LIN {X 20.739,Y -41.059,Z -74.568,A -90.000,B 90.000,C 0.000} C_DIS
LIN {X 20.794,Y -41.067,Z -74.409,A -90.000,B 90.000,C 0.000} C_DIS
LIN {X 20.845,Y -41.076,Z -74.290,A -90.000,B 90.000,C 0.000} C_DIS
LIN {X 20.887,Y -41.080,Z -74.206,A -90.000,B 90.000,C 0.000} C_DIS
LIN {X 20.922,Y -41.083,Z -74.143,A -90.000,B 90.000,C 0.000} C_DIS
LIN {X 20.977,Y -41.084,Z -74.055,A -90.000,B 90.000,C 0.000} C_DIS
LIN {X 21.019,Y -41.085,Z -73.993,A -90.000,B 90.000,C 0.000} C_DIS
LIN {X 21.124,Y -41.081,Z -73.850,A -90.000,B 90.000,C 0.000} C_DIS
LIN {X 21.182,Y -41.076,Z -73.781,A -90.000,B 90.000,C 0.000} C_DIS
LIN {X 21.231,Y -41.072,Z -73.726,A -90.000,B 90.000,C 0.000} C_DIS
LIN {X 21.448,Y -41.048,Z -73.510,A -90.000,B 90.000,C 0.000} C_DIS
LIN {X 21.548,Y -41.035,Z -73.423,A -90.000,B 90.000,C 0.000} C_DIS
LIN {X 21.638,Y -41.027,Z -73.353,A -90.000,B 90.000,C 0.000} C_DIS
LIN {X 21.731,Y -41.021,Z -73.289,A -90.000,B 90.000,C 0.000} C_DIS
LIN {X 21.845,Y -41.016,Z -73.219,A -90.000,B 90.000,C 0.000} C_DIS
LIN {X 22.045,Y -41.002,Z -73.109,A -90.000,B 90.000,C 0.000} C_DIS
LIN {X 22.194,Y -40.983,Z -73.040,A -90.000,B 90.000,C 0.000} C_DIS
LIN {X 22.361,Y -40.964,Z -72.980,A -90.000,B 90.000,C 0.000} C_DIS
LIN {X 22.407,Y -40.959,Z -72.966,A -90.000,B 90.000,C 0.000} C_DIS
LIN {X 22.608,Y -40.941,Z -72.918,A -90.000,B 90.000,C 0.000} C_DIS
LIN {X 22.750,Y -40.923,Z -72.888,A -90.000,B 90.000,C 0.000} C_DIS
LIN {X 22.851,Y -40.911,Z -72.872,A -90.000,B 90.000,C 0.000} C_DIS
LIN {X 22.918,Y -40.901,Z -72.865,A -90.000,B 90.000,C 0.000} C_DIS
LIN {X 22.991,Y -40.890,Z -72.860,A -90.000,B 90.000,C 0.000} C_DIS
LIN {X 23.121,Y -40.871,Z -72.857,A -90.000,B 90.000,C 0.000} C_DIS
LIN {X 23.421,Y -40.816,Z -72.816,A -90.000,B 90.000,C 0.000} C_DIS
LIN {X 23.607,Y -40.785,Z -72.800,A -90.000,B 90.000,C 0.000} C_DIS
LIN {X 23.837,Y -40.743,Z -72.806,A -90.000,B 90.000,C 0.000} C_DIS
LIN {X 24.098,Y -40.703,Z -72.831,A -90.000,B 90.000,C 0.000} C_DIS
LIN {X 24.287,Y -40.682,Z -72.862,A -90.000,B 90.000,C 0.000} C_DIS
LIN {X 24.457,Y -40.670,Z -72.906,A -90.000,B 90.000,C 0.000} C_DIS
LIN {X 24.895,Y -40.649,Z -73.037,A -90.000,B 90.000,C 0.000} C_DIS
LIN {X 24.984,Y -40.642,Z -73.064,A -90.000,B 90.000,C 0.000} C_DIS
LIN {X 25.233,Y -40.629,Z -73.149,A -90.000,B 90.000,C 0.000} C_DIS
LIN {X 25.886,Y -40.603,Z -73.389,A -90.000,B 90.000,C 0.000} C_DIS
LIN {X 26.129,Y -40.642,Z -73.460,A -90.000,B 90.000,C 0.000} C_DIS
LIN {X 26.235,Y -40.654,Z -73.492,A -90.000,B 90.000,C 0.000} C_DIS
LIN {X 26.356,Y -40.664,Z -73.532,A -90.000,B 90.000,C 0.000} C_DIS
LIN {X 26.477,Y -40.671,Z -73.577,A -90.000,B 90.000,C 0.000} C_DIS
LIN {X 26.624,Y -40.675,Z -73.643,A -90.000,B 90.000,C 0.000} C_DIS
LIN {X 26.712,Y -40.674,Z -73.692,A -90.000,B 90.000,C 0.000} C_DIS
LIN {X 26.777,Y -40.673,Z -73.731,A -90.000,B 90.000,C 0.000} C_DIS
LIN {X 27.152,Y -40.658,Z -73.985,A -90.000,B 90.000,C 0.000} C_DIS
LIN {X 27.234,Y -40.655,Z -74.042,A -90.000,B 90.000,C 0.000} C_DIS
LIN {X 27.334,Y -40.665,Z -74.106,A -90.000,B 90.000,C 0.000} C_DIS
LIN {X 27.515,Y -40.693,Z -74.240,A -90.000,B 90.000,C 0.000} C_DIS
LIN {X 27.742,Y -40.737,Z -74.427,A -90.000,B 90.000,C 0.000} C_DIS
LIN {X 28.067,Y -40.769,Z -74.619,A -90.000,B 90.000,C 0.000} C_DIS
LIN {X 28.270,Y -40.787,Z -74.741,A -90.000,B 90.000,C 0.000} C_DIS
LIN {X 28.484,Y -40.804,Z -74.883,A -90.000,B 90.000,C 0.000} C_DIS
LIN {X 28.589,Y -40.816,Z -74.962,A -90.000,B 90.000,C 0.000} C_DIS
LIN {X 28.701,Y -40.830,Z -75.051,A -90.000,B 90.000,C 0.000} C_DIS
LIN {X 28.816,Y -40.850,Z -75.156,A -90.000,B 90.000,C 0.000} C_DIS
LIN {X 28.899,Y -40.868,Z -75.243,A -90.000,B 90.000,C 0.000} C_DIS
LIN {X 29.007,Y -40.894,Z -75.364,A -90.000,B 90.000,C 0.000} C_DIS
LIN {X 29.056,Y -40.902,Z -75.422,A -90.000,B 90.000,C 0.000} C_DIS
LIN {X 29.140,Y -40.918,Z -75.531,A -90.000,B 90.000,C 0.000} C_DIS
LIN {X 29.065,Y -40.889,Z -75.375,A -90.000,B 90.000,C 0.000} C_DIS
LIN {X 29.035,Y -40.867,Z -75.304,A -90.000,B 90.000,C 0.000} C_DIS
LIN {X 28.987,Y -40.823,Z -75.163,A -90.000,B 90.000,C 0.000} C_DIS
LIN {X 28.912,Y -40.733,Z -74.888,A -90.000,B 90.000,C 0.000} C_DIS
LIN {X 28.896,Y -40.706,Z -74.820,A -90.000,B 90.000,C 0.000} C_DIS
LIN {X 28.875,Y -40.655,Z -74.711,A -90.000,B 90.000,C 0.000} C_DIS
LIN {X 28.863,Y -40.607,Z -74.612,A -90.000,B 90.000,C 0.000} C_DIS
LIN {X 28.857,Y -40.573,Z -74.542,A -90.000,B 90.000,C 0.000} C_DIS
LIN {X 28.785,Y -40.606,Z -74.333,A -90.000,B 90.000,C 0.000} C_DIS
LIN {X 28.697,Y -40.642,Z -74.065,A -90.000,B 90.000,C 0.000} C_DIS
LIN {X 28.660,Y -40.658,Z -73.938,A -90.000,B 90.000,C 0.000} C_DIS
LIN {X 28.633,Y -40.670,Z -73.800,A -90.000,B 90.000,C 0.000} C_DIS
LIN {X 28.563,Y -40.700,Z -73.393,A -90.000,B 90.000,C 0.000} C_DIS
LIN {X 28.554,Y -40.704,Z -73.311,A -90.000,B 90.000,C 0.000} C_DIS
LIN {X 28.534,Y -40.707,Z -73.108,A -90.000,B 90.000,C 0.000} C_DIS
LIN {X 28.507,Y -40.700,Z -72.788,A -90.000,B 90.000,C 0.000} C_DIS
LIN {X 28.500,Y -40.696,Z -72.665,A -90.000,B 90.000,C 0.000} C_DIS
LIN {X 28.496,Y -40.692,Z -72.535,A -90.000,B 90.000,C 0.000} C_DIS
LIN {X 28.495,Y -40.688,Z -72.486,A -90.000,B 90.000,C 0.000} C_DIS
LIN {X 28.495,Y -40.679,Z -72.413,A -90.000,B 90.000,C 0.000} C_DIS
LIN {X 28.493,Y -40.678,Z -72.374,A -90.000,B 90.000,C 0.000} C_DIS
LIN {X 28.493,Y -40.673,Z -72.333,A -90.000,B 90.000,C 0.000} C_DIS
LIN {X 28.491,Y -40.602,Z -71.772,A -90.000,B 90.000,C 0.000} C_DIS
LIN {X 28.496,Y -40.578,Z -71.671,A -90.000,B 90.000,C 0.000} C_DIS
LIN {X 28.513,Y -40.524,Z -71.446,A -90.000,B 90.000,C 0.000} C_DIS
LIN {X 28.522,Y -40.503,Z -71.363,A -90.000,B 90.000,C 0.000} C_DIS
LIN {X 28.535,Y -40.479,Z -71.269,A -90.000,B 90.000,C 0.000} C_DIS
LIN {X 28.558,Y -40.435,Z -71.147,A -90.000,B 90.000,C 0.000} C_DIS
LIN {X 28.608,Y -40.348,Z -70.924,A -90.000,B 90.000,C 0.000} C_DIS
LIN {X 28.637,Y -40.307,Z -70.822,A -90.000,B 90.000,C 0.000} C_DIS
LIN {X 28.684,Y -40.248,Z -70.684,A -90.000,B 90.000,C 0.000} C_DIS
LIN {X 28.761,Y -40.153,Z -70.522,A -90.000,B 90.000,C 0.000} C_DIS
LIN {X 28.872,Y -40.031,Z -70.321,A -90.000,B 90.000,C 0.000} C_DIS
LIN {X 28.886,Y -40.016,Z -70.298,A -90.000,B 90.000,C 0.000} C_DIS
LIN {X 28.903,Y -39.999,Z -70.278,A -90.000,B 90.000,C 0.000} C_DIS
LIN {X 28.971,Y -39.931,Z -70.206,A -90.000,B 90.000,C 0.000} C_DIS
LIN {X 29.041,Y -39.869,Z -70.144,A -90.000,B 90.000,C 0.000} C_DIS
LIN {X 29.042,Y -39.892,Z -69.943,A -90.000,B 90.000,C 0.000} C_DIS
LIN {X 29.046,Y -39.912,Z -69.756,A -90.000,B 90.000,C 0.000} C_DIS
LIN {X 29.061,Y -39.961,Z -69.383,A -90.000,B 90.000,C 0.000} C_DIS
LIN {X 29.065,Y -39.977,Z -69.251,A -90.000,B 90.000,C 0.000} C_DIS
LIN {X 29.040,Y -39.961,Z -69.052,A -90.000,B 90.000,C 0.000} C_DIS
LIN {X 29.024,Y -39.953,Z -68.893,A -90.000,B 90.000,C 0.000} C_DIS
LIN {X 29.017,Y -39.952,Z -68.804,A -90.000,B 90.000,C 0.000} C_DIS
LIN {X 29.002,Y -39.952,Z -68.566,A -90.000,B 90.000,C 0.000} C_DIS
LIN {X 28.985,Y -39.943,Z -68.293,A -90.000,B 90.000,C 0.000} C_DIS
LIN {X 28.973,Y -39.937,Z -68.071,A -90.000,B 90.000,C 0.000} C_DIS
LIN {X 28.934,Y -39.926,Z -67.437,A -90.000,B 90.000,C 0.000} C_DIS
LIN {X 28.921,Y -39.924,Z -67.208,A -90.000,B 90.000,C 0.000} C_DIS
LIN {X 28.917,Y -39.922,Z -67.103,A -90.000,B 90.000,C 0.000} C_DIS
LIN {X 28.915,Y -39.923,Z -66.972,A -90.000,B 90.000,C 0.000} C_DIS
LIN {X 28.917,Y -39.946,Z -66.272,A -90.000,B 90.000,C 0.000} C_DIS
LIN {X 28.925,Y -39.969,Z -65.802,A -90.000,B 90.000,C 0.000} C_DIS
LIN {X 28.936,Y -39.980,Z -65.477,A -90.000,B 90.000,C 0.000} C_DIS
LIN {X 28.952,Y -39.998,Z -65.100,A -90.000,B 90.000,C 0.000} C_DIS
LIN {X 28.961,Y -40.008,Z -64.964,A -90.000,B 90.000,C 0.000} C_DIS
LIN {X 28.991,Y -40.040,Z -64.705,A -90.000,B 90.000,C 0.000} C_DIS
LIN {X 29.056,Y -40.094,Z -64.224,A -90.000,B 90.000,C 0.000} C_DIS
LIN {X 29.097,Y -40.123,Z -63.947,A -90.000,B 90.000,C 0.000} C_DIS
LIN {X 29.164,Y -40.154,Z -63.594,A -90.000,B 90.000,C 0.000} C_DIS
LIN {X 29.181,Y -40.164,Z -63.517,A -90.000,B 90.000,C 0.000} C_DIS
LIN {X 29.246,Y -40.202,Z -63.255,A -90.000,B 90.000,C 0.000} C_DIS
LIN {X 29.278,Y -40.220,Z -63.112,A -90.000,B 90.000,C 0.000} C_DIS
LIN {X 29.318,Y -40.233,Z -62.982,A -90.000,B 90.000,C 0.000} C_DIS
LIN {X 29.371,Y -40.252,Z -62.818,A -90.000,B 90.000,C 0.000} C_DIS
LIN {X 29.470,Y -40.290,Z -62.526,A -90.000,B 90.000,C 0.000} C_DIS
LIN {X 29.513,Y -40.308,Z -62.410,A -90.000,B 90.000,C 0.000} C_DIS
LIN {X 29.558,Y -40.330,Z -62.304,A -90.000,B 90.000,C 0.000} C_DIS
LIN {X 29.722,Y -40.380,Z -61.991,A -90.000,B 90.000,C 0.000} C_DIS
LIN {X 29.790,Y -40.400,Z -61.875,A -90.000,B 90.000,C 0.000} C_DIS
LIN {X 29.906,Y -40.431,Z -61.702,A -90.000,B 90.000,C 0.000} C_DIS
LIN {X 30.022,Y -40.458,Z -61.534,A -90.000,B 90.000,C 0.000} C_DIS
LIN {X 30.098,Y -40.470,Z -61.437,A -90.000,B 90.000,C 0.000} C_DIS
LIN {X 30.199,Y -40.487,Z -61.317,A -90.000,B 90.000,C 0.000} C_DIS
LIN {X 30.265,Y -40.494,Z -61.242,A -90.000,B 90.000,C 0.000} C_DIS
LIN {X 30.445,Y -40.400,Z -60.703,A -90.000,B 90.000,C 0.000} C_DIS
LIN {X 30.536,Y -40.349,Z -60.445,A -90.000,B 90.000,C 0.000} C_DIS
LIN {X 30.632,Y -40.305,Z -60.205,A -90.000,B 90.000,C 0.000} C_DIS
LIN {X 30.748,Y -40.248,Z -59.942,A -90.000,B 90.000,C 0.000} C_DIS
LIN {X 30.826,Y -40.210,Z -59.773,A -90.000,B 90.000,C 0.000} C_DIS
LIN {X 30.903,Y -40.172,Z -59.615,A -90.000,B 90.000,C 0.000} C_DIS
LIN {X 30.938,Y -40.153,Z -59.545,A -90.000,B 90.000,C 0.000} C_DIS
LIN {X 31.044,Y -40.095,Z -59.356,A -90.000,B 90.000,C 0.000} C_DIS
LIN {X 31.169,Y -40.028,Z -59.149,A -90.000,B 90.000,C 0.000} C_DIS
LIN {X 31.259,Y -39.978,Z -59.017,A -90.000,B 90.000,C 0.000} C_DIS
LIN {X 31.430,Y -39.885,Z -58.777,A -90.000,B 90.000,C 0.000} C_DIS
LIN {X 31.622,Y -39.782,Z -58.547,A -90.000,B 90.000,C 0.000} C_DIS
LIN {X 31.743,Y -39.722,Z -58.414,A -90.000,B 90.000,C 0.000} C_DIS
LIN {X 31.849,Y -39.675,Z -58.309,A -90.000,B 90.000,C 0.000} C_DIS
LIN {X 31.940,Y -39.637,Z -58.230,A -90.000,B 90.000,C 0.000} C_DIS
LIN {X 32.000,Y -39.612,Z -58.182,A -90.000,B 90.000,C 0.000} C_DIS
LIN {X 32.051,Y -39.624,Z -57.993,A -90.000,B 90.000,C 0.000} C_DIS
LIN {X 32.124,Y -39.645,Z -57.729,A -90.000,B 90.000,C 0.000} C_DIS
LIN {X 32.237,Y -39.661,Z -57.406,A -90.000,B 90.000,C 0.000} C_DIS
LIN {X 32.279,Y -39.668,Z -57.289,A -90.000,B 90.000,C 0.000} C_DIS
LIN {X 32.419,Y -39.706,Z -56.914,A -90.000,B 90.000,C 0.000} C_DIS
LIN {X 32.507,Y -39.732,Z -56.679,A -90.000,B 90.000,C 0.000} C_DIS
LIN {X 32.616,Y -39.765,Z -56.387,A -90.000,B 90.000,C 0.000} C_DIS
LIN {X 32.780,Y -39.791,Z -56.009,A -90.000,B 90.000,C 0.000} C_DIS
LIN {X 32.795,Y -39.792,Z -55.977,A -90.000,B 90.000,C 0.000} C_DIS
LIN {X 32.962,Y -39.810,Z -55.645,A -90.000,B 90.000,C 0.000} C_DIS
LIN {X 33.054,Y -39.815,Z -55.481,A -90.000,B 90.000,C 0.000} C_DIS
LIN {X 33.192,Y -39.830,Z -55.249,A -90.000,B 90.000,C 0.000} C_DIS
LIN {X 33.254,Y -39.840,Z -55.140,A -90.000,B 90.000,C 0.000} C_DIS
LIN {X 33.328,Y -39.853,Z -55.016,A -90.000,B 90.000,C 0.000} C_DIS
LIN {X 33.395,Y -39.866,Z -54.907,A -90.000,B 90.000,C 0.000} C_DIS
LIN {X 33.569,Y -39.902,Z -54.644,A -90.000,B 90.000,C 0.000} C_DIS
LIN {X 33.738,Y -39.918,Z -54.422,A -90.000,B 90.000,C 0.000} C_DIS
LIN {X 33.790,Y -39.921,Z -54.349,A -90.000,B 90.000,C 0.000} C_DIS
LIN {X 33.978,Y -39.939,Z -54.105,A -90.000,B 90.000,C 0.000} C_DIS
LIN {X 34.106,Y -39.942,Z -53.956,A -90.000,B 90.000,C 0.000} C_DIS
LIN {X 34.227,Y -39.950,Z -53.825,A -90.000,B 90.000,C 0.000} C_DIS
LIN {X 34.393,Y -39.967,Z -53.656,A -90.000,B 90.000,C 0.000} C_DIS
LIN {X 34.458,Y -39.977,Z -53.586,A -90.000,B 90.000,C 0.000} C_DIS
LIN {X 34.610,Y -39.992,Z -53.434,A -90.000,B 90.000,C 0.000} C_DIS
LIN {X 34.752,Y -40.008,Z -53.298,A -90.000,B 90.000,C 0.000} C_DIS
LIN {X 34.881,Y -40.012,Z -53.188,A -90.000,B 90.000,C 0.000} C_DIS
LIN {X 35.056,Y -40.015,Z -53.038,A -90.000,B 90.000,C 0.000} C_DIS
LIN {X 35.286,Y -40.009,Z -52.849,A -90.000,B 90.000,C 0.000} C_DIS
LIN {X 35.372,Y -40.009,Z -52.781,A -90.000,B 90.000,C 0.000} C_DIS
LIN {X 35.531,Y -40.015,Z -52.664,A -90.000,B 90.000,C 0.000} C_DIS
LIN {X 35.642,Y -40.023,Z -52.579,A -90.000,B 90.000,C 0.000} C_DIS
LIN {X 35.671,Y -40.025,Z -52.557,A -90.000,B 90.000,C 0.000} C_DIS
LIN {X 35.763,Y -40.025,Z -52.495,A -90.000,B 90.000,C 0.000} C_DIS
LIN {X 35.882,Y -40.031,Z -52.421,A -90.000,B 90.000,C 0.000} C_DIS
LIN {X 36.011,Y -40.041,Z -52.346,A -90.000,B 90.000,C 0.000} C_DIS
LIN {X 36.370,Y -40.043,Z -52.163,A -90.000,B 90.000,C 0.000} C_DIS
LIN {X 36.876,Y -40.035,Z -51.920,A -90.000,B 90.000,C 0.000} C_DIS
LIN {X 37.014,Y -40.034,Z -51.853,A -90.000,B 90.000,C 0.000} C_DIS
LIN {X 37.118,Y -40.036,Z -51.804,A -90.000,B 90.000,C 0.000} C_DIS
LIN {X 37.496,Y -40.037,Z -51.667,A -90.000,B 90.000,C 0.000} C_DIS
LIN {X 37.531,Y -40.035,Z -51.656,A -90.000,B 90.000,C 0.000} C_DIS
LIN {X 37.760,Y -40.029,Z -51.596,A -90.000,B 90.000,C 0.000} C_DIS
LIN {X 37.885,Y -40.030,Z -51.568,A -90.000,B 90.000,C 0.000} C_DIS
LIN {X 38.118,Y -40.025,Z -51.523,A -90.000,B 90.000,C 0.000} C_DIS
LIN {X 38.467,Y -40.023,Z -51.460,A -90.000,B 90.000,C 0.000} C_DIS
LIN {X 38.781,Y -40.023,Z -51.405,A -90.000,B 90.000,C 0.000} C_DIS
LIN {X 38.981,Y -40.016,Z -51.377,A -90.000,B 90.000,C 0.000} C_DIS
LIN {X 39.176,Y -40.011,Z -51.350,A -90.000,B 90.000,C 0.000} C_DIS
LIN {X 39.568,Y -39.990,Z -51.337,A -90.000,B 90.000,C 0.000} C_DIS
LIN {X 39.615,Y -39.985,Z -51.337,A -90.000,B 90.000,C 0.000} C_DIS
LIN {X 39.826,Y -39.975,Z -51.345,A -90.000,B 90.000,C 0.000} C_DIS
LIN {X 40.191,Y -39.968,Z -51.370,A -90.000,B 90.000,C 0.000} C_DIS
LIN {X 40.277,Y -39.968,Z -51.378,A -90.000,B 90.000,C 0.000} C_DIS
LIN {X 40.534,Y -39.973,Z -51.405,A -90.000,B 90.000,C 0.000} C_DIS
LIN {X 41.084,Y -39.977,Z -51.468,A -90.000,B 90.000,C 0.000} C_DIS
LIN {X 41.333,Y -39.964,Z -51.510,A -90.000,B 90.000,C 0.000} C_DIS
LIN {X 41.488,Y -39.958,Z -51.538,A -90.000,B 90.000,C 0.000} C_DIS
LIN {X 41.818,Y -39.925,Z -51.619,A -90.000,B 90.000,C 0.000} C_DIS
LIN {X 41.982,Y -39.914,Z -51.665,A -90.000,B 90.000,C 0.000} C_DIS
LIN {X 42.309,Y -39.902,Z -51.767,A -90.000,B 90.000,C 0.000} C_DIS
LIN {X 42.366,Y -39.899,Z -51.786,A -90.000,B 90.000,C 0.000} C_DIS
LIN {X 42.524,Y -39.895,Z -51.844,A -90.000,B 90.000,C 0.000} C_DIS
LIN {X 42.767,Y -39.896,Z -51.941,A -90.000,B 90.000,C 0.000} C_DIS
LIN {X 42.994,Y -39.896,Z -52.034,A -90.000,B 90.000,C 0.000} C_DIS
LIN {X 43.316,Y -39.884,Z -52.180,A -90.000,B 90.000,C 0.000} C_DIS
LIN {X 44.072,Y -39.861,Z -52.532,A -90.000,B 90.000,C 0.000} C_DIS
LIN {X 44.285,Y -39.859,Z -52.637,A -90.000,B 90.000,C 0.000} C_DIS
LIN {X 44.360,Y -39.858,Z -52.676,A -90.000,B 90.000,C 0.000} C_DIS
LIN {X 44.589,Y -39.862,Z -52.784,A -90.000,B 90.000,C 0.000} C_DIS
LIN {X 44.667,Y -39.865,Z -52.822,A -90.000,B 90.000,C 0.000} C_DIS
LIN {X 45.073,Y -39.887,Z -53.030,A -90.000,B 90.000,C 0.000} C_DIS
LIN {X 45.289,Y -39.893,Z -53.147,A -90.000,B 90.000,C 0.000} C_DIS
LIN {X 45.630,Y -39.938,Z -53.295,A -90.000,B 90.000,C 0.000} C_DIS
LIN {X 45.753,Y -39.958,Z -53.355,A -90.000,B 90.000,C 0.000} C_DIS
LIN {X 45.891,Y -40.000,Z -53.405,A -90.000,B 90.000,C 0.000} C_DIS
LIN {X 46.070,Y -40.052,Z -53.469,A -90.000,B 90.000,C 0.000} C_DIS
LIN {X 46.416,Y -40.159,Z -53.596,A -90.000,B 90.000,C 0.000} C_DIS
LIN {X 46.521,Y -40.196,Z -53.634,A -90.000,B 90.000,C 0.000} C_DIS
LIN {X 46.624,Y -40.202,Z -53.629,A -90.000,B 90.000,C 0.000} C_DIS
LIN {X 47.199,Y -40.201,Z -53.555,A -90.000,B 90.000,C 0.000} C_DIS
LIN {X 47.743,Y -40.204,Z -53.481,A -90.000,B 90.000,C 0.000} C_DIS
LIN {X 47.853,Y -40.203,Z -53.471,A -90.000,B 90.000,C 0.000} C_DIS
LIN {X 48.141,Y -40.205,Z -53.451,A -90.000,B 90.000,C 0.000} C_DIS
LIN {X 48.262,Y -40.202,Z -53.446,A -90.000,B 90.000,C 0.000} C_DIS
LIN {X 49.295,Y -40.205,Z -53.453,A -90.000,B 90.000,C 0.000} C_DIS
LIN {X 49.748,Y -40.210,Z -53.452,A -90.000,B 90.000,C 0.000} C_DIS
LIN {X 49.874,Y -40.208,Z -53.455,A -90.000,B 90.000,C 0.000} C_DIS
LIN {X 49.991,Y -40.207,Z -53.460,A -90.000,B 90.000,C 0.000} C_DIS
LIN {X 50.126,Y -40.208,Z -53.470,A -90.000,B 90.000,C 0.000} C_DIS
LIN {X 50.402,Y -40.194,Z -53.502,A -90.000,B 90.000,C 0.000} C_DIS
LIN {X 50.496,Y -40.192,Z -53.517,A -90.000,B 90.000,C 0.000} C_DIS
LIN {X 50.915,Y -40.174,Z -53.621,A -90.000,B 90.000,C 0.000} C_DIS
LIN {X 51.112,Y -40.173,Z -53.679,A -90.000,B 90.000,C 0.000} C_DIS
LIN {X 51.548,Y -40.185,Z -53.827,A -90.000,B 90.000,C 0.000} C_DIS
LIN {X 51.911,Y -40.190,Z -53.945,A -90.000,B 90.000,C 0.000} C_DIS
LIN {X 52.247,Y -40.200,Z -54.051,A -90.000,B 90.000,C 0.000} C_DIS
LIN {X 52.651,Y -40.202,Z -54.184,A -90.000,B 90.000,C 0.000} C_DIS
LIN {X 52.804,Y -40.191,Z -54.243,A -90.000,B 90.000,C 0.000} C_DIS
LIN {X 52.991,Y -40.182,Z -54.320,A -90.000,B 90.000,C 0.000} C_DIS
LIN {X 53.182,Y -40.162,Z -54.407,A -90.000,B 90.000,C 0.000} C_DIS
LIN {X 53.255,Y -40.156,Z -54.442,A -90.000,B 90.000,C 0.000} C_DIS
LIN {X 53.347,Y -40.152,Z -54.489,A -90.000,B 90.000,C 0.000} C_DIS
LIN {X 53.681,Y -40.126,Z -54.694,A -90.000,B 90.000,C 0.000} C_DIS
LIN {X 53.815,Y -40.120,Z -54.783,A -90.000,B 90.000,C 0.000} C_DIS
LIN {X 54.184,Y -40.113,Z -55.043,A -90.000,B 90.000,C 0.000} C_DIS
LIN {X 54.325,Y -40.115,Z -55.151,A -90.000,B 90.000,C 0.000} C_DIS
LIN {X 55.267,Y -40.165,Z -55.920,A -90.000,B 90.000,C 0.000} C_DIS
LIN {X 55.556,Y -40.166,Z -56.169,A -90.000,B 90.000,C 0.000} C_DIS
LIN {X 55.654,Y -40.159,Z -56.260,A -90.000,B 90.000,C 0.000} C_DIS
LIN {X 56.087,Y -40.112,Z -56.658,A -90.000,B 90.000,C 0.000} C_DIS
LIN {X 56.396,Y -40.082,Z -56.955,A -90.000,B 90.000,C 0.000} C_DIS
LIN {X 56.497,Y -40.075,Z -57.058,A -90.000,B 90.000,C 0.000} C_DIS
LIN {X 56.789,Y -40.071,Z -57.390,A -90.000,B 90.000,C 0.000} C_DIS
LIN {X 57.498,Y -40.083,Z -58.244,A -90.000,B 90.000,C 0.000} C_DIS
LIN {X 57.586,Y -40.088,Z -58.356,A -90.000,B 90.000,C 0.000} C_DIS
LIN {X 57.748,Y -40.101,Z -58.574,A -90.000,B 90.000,C 0.000} C_DIS
LIN {X 58.128,Y -40.098,Z -59.131,A -90.000,B 90.000,C 0.000} C_DIS
LIN {X 58.196,Y -40.099,Z -59.233,A -90.000,B 90.000,C 0.000} C_DIS
LIN {X 58.620,Y -40.116,Z -59.903,A -90.000,B 90.000,C 0.000} C_DIS
LIN {X 58.662,Y -40.119,Z -59.972,A -90.000,B 90.000,C 0.000} C_DIS
LIN {X 58.840,Y -40.136,Z -60.275,A -90.000,B 90.000,C 0.000} C_DIS
LIN {X 58.923,Y -40.146,Z -60.421,A -90.000,B 90.000,C 0.000} C_DIS
LIN {X 59.311,Y -40.200,Z -61.118,A -90.000,B 90.000,C 0.000} C_DIS
LIN {X 59.694,Y -40.209,Z -61.875,A -90.000,B 90.000,C 0.000} C_DIS
LIN {X 60.121,Y -40.201,Z -62.753,A -90.000,B 90.000,C 0.000} C_DIS
LIN {X 60.188,Y -40.203,Z -62.905,A -90.000,B 90.000,C 0.000} C_DIS
LIN {X 60.318,Y -40.217,Z -63.231,A -90.000,B 90.000,C 0.000} C_DIS
LIN {X 60.363,Y -40.224,Z -63.352,A -90.000,B 90.000,C 0.000} C_DIS
LIN {X 60.483,Y -40.252,Z -63.707,A -90.000,B 90.000,C 0.000} C_DIS
LIN {X 60.795,Y -40.313,Z -64.586,A -90.000,B 90.000,C 0.000} C_DIS
LIN {X 60.899,Y -40.321,Z -64.906,A -90.000,B 90.000,C 0.000} C_DIS
LIN {X 60.945,Y -40.321,Z -65.054,A -90.000,B 90.000,C 0.000} C_DIS
LIN {X 60.977,Y -40.318,Z -65.143,A -90.000,B 90.000,C 0.000} C_DIS
LIN {X 61.064,Y -40.318,Z -65.373,A -90.000,B 90.000,C 0.000} C_DIS
LIN {X 61.169,Y -40.325,Z -65.652,A -90.000,B 90.000,C 0.000} C_DIS
LIN {X 61.296,Y -40.341,Z -66.024,A -90.000,B 90.000,C 0.000} C_DIS
LIN {X 61.364,Y -40.358,Z -66.262,A -90.000,B 90.000,C 0.000} C_DIS
LIN {X 61.404,Y -40.375,Z -66.389,A -90.000,B 90.000,C 0.000} C_DIS
LIN {X 61.437,Y -40.392,Z -66.506,A -90.000,B 90.000,C 0.000} C_DIS
LIN {X 61.453,Y -40.404,Z -66.578,A -90.000,B 90.000,C 0.000} C_DIS
LIN {X 61.531,Y -40.476,Z -66.992,A -90.000,B 90.000,C 0.000} C_DIS
LIN {X 61.586,Y -40.495,Z -67.165,A -90.000,B 90.000,C 0.000} C_DIS
LIN {X 61.667,Y -40.510,Z -67.445,A -90.000,B 90.000,C 0.000} C_DIS
LIN {X 61.699,Y -40.513,Z -67.560,A -90.000,B 90.000,C 0.000} C_DIS
LIN {X 61.837,Y -40.496,Z -67.876,A -90.000,B 90.000,C 0.000} C_DIS
LIN {X 61.967,Y -40.504,Z -68.147,A -90.000,B 90.000,C 0.000} C_DIS
LIN {X 62.039,Y -40.513,Z -68.314,A -90.000,B 90.000,C 0.000} C_DIS
LIN {X 62.081,Y -40.524,Z -68.434,A -90.000,B 90.000,C 0.000} C_DIS
LIN {X 62.184,Y -40.557,Z -68.767,A -90.000,B 90.000,C 0.000} C_DIS
LIN {X 62.212,Y -40.570,Z -68.877,A -90.000,B 90.000,C 0.000} C_DIS
LIN {X 62.235,Y -40.594,Z -68.976,A -90.000,B 90.000,C 0.000} C_DIS
LIN {X 62.254,Y -40.619,Z -69.076,A -90.000,B 90.000,C 0.000} C_DIS
LIN {X 62.309,Y -40.686,Z -69.445,A -90.000,B 90.000,C 0.000} C_DIS
LIN {X 62.414,Y -40.703,Z -69.674,A -90.000,B 90.000,C 0.000} C_DIS
LIN {X 62.507,Y -40.705,Z -69.884,A -90.000,B 90.000,C 0.000} C_DIS
LIN {X 62.546,Y -40.702,Z -69.941,A -90.000,B 90.000,C 0.000} C_DIS
LIN {X 62.691,Y -40.685,Z -70.152,A -90.000,B 90.000,C 0.000} C_DIS
LIN {X 62.756,Y -40.680,Z -70.263,A -90.000,B 90.000,C 0.000} C_DIS
LIN {X 62.845,Y -40.673,Z -70.420,A -90.000,B 90.000,C 0.000} C_DIS
LIN {X 62.863,Y -40.675,Z -70.449,A -90.000,B 90.000,C 0.000} C_DIS
LIN {X 62.930,Y -40.686,Z -70.567,A -90.000,B 90.000,C 0.000} C_DIS
LIN {X 63.000,Y -40.702,Z -70.713,A -90.000,B 90.000,C 0.000} C_DIS
LIN {X 63.052,Y -40.720,Z -70.847,A -90.000,B 90.000,C 0.000} C_DIS
LIN {X 63.132,Y -40.750,Z -71.061,A -90.000,B 90.000,C 0.000} C_DIS
LIN {X 63.168,Y -40.767,Z -71.171,A -90.000,B 90.000,C 0.000} C_DIS
LIN {X 63.239,Y -40.802,Z -71.412,A -90.000,B 90.000,C 0.000} C_DIS
LIN {X 63.274,Y -40.828,Z -71.524,A -90.000,B 90.000,C 0.000} C_DIS
LIN {X 63.301,Y -40.854,Z -71.628,A -90.000,B 90.000,C 0.000} C_DIS
LIN {X 63.311,Y -40.863,Z -71.679,A -90.000,B 90.000,C 0.000} C_DIS
LIN {X 63.341,Y -40.893,Z -71.848,A -90.000,B 90.000,C 0.000} C_DIS
LIN {X 63.368,Y -40.935,Z -72.081,A -90.000,B 90.000,C 0.000} C_DIS
LIN {X 63.452,Y -40.946,Z -72.217,A -90.000,B 90.000,C 0.000} C_DIS
LIN {X 63.786,Y -40.929,Z -72.492,A -90.000,B 90.000,C 0.000} C_DIS
LIN {X 64.167,Y -40.899,Z -72.809,A -90.000,B 90.000,C 0.000} C_DIS
LIN {X 64.307,Y -40.889,Z -72.928,A -90.000,B 90.000,C 0.000} C_DIS
LIN {X 64.496,Y -40.878,Z -73.127,A -90.000,B 90.000,C 0.000} C_DIS
LIN {X 64.618,Y -40.888,Z -73.269,A -90.000,B 90.000,C 0.000} C_DIS
LIN {X 64.696,Y -40.895,Z -73.366,A -90.000,B 90.000,C 0.000} C_DIS
LIN {X 64.807,Y -40.900,Z -73.511,A -90.000,B 90.000,C 0.000} C_DIS
LIN {X 65.561,Y -40.793,Z -73.791,A -90.000,B 90.000,C 0.000} C_DIS
LIN {X 65.942,Y -40.738,Z -73.935,A -90.000,B 90.000,C 0.000} C_DIS
LIN {X 65.969,Y -40.737,Z -73.944,A -90.000,B 90.000,C 0.000} C_DIS
LIN {X 66.194,Y -40.728,Z -74.039,A -90.000,B 90.000,C 0.000} C_DIS
LIN {X 66.937,Y -40.714,Z -74.403,A -90.000,B 90.000,C 0.000} C_DIS
LIN {X 67.134,Y -40.704,Z -74.502,A -90.000,B 90.000,C 0.000} C_DIS
LIN {X 67.285,Y -40.696,Z -74.582,A -90.000,B 90.000,C 0.000} C_DIS
LIN {X 67.764,Y -40.679,Z -74.857,A -90.000,B 90.000,C 0.000} C_DIS
LIN {X 67.835,Y -40.677,Z -74.900,A -90.000,B 90.000,C 0.000} C_DIS
LIN {X 67.911,Y -40.676,Z -74.949,A -90.000,B 90.000,C 0.000} C_DIS
LIN {X 68.130,Y -40.678,Z -75.105,A -90.000,B 90.000,C 0.000} C_DIS
LIN {X 68.280,Y -40.682,Z -75.223,A -90.000,B 90.000,C 0.000} C_DIS
LIN {X 68.897,Y -40.724,Z -75.781,A -90.000,B 90.000,C 0.000} C_DIS
LIN {X 68.986,Y -40.724,Z -75.865,A -90.000,B 90.000,C 0.000} C_DIS
LIN {X 69.052,Y -40.732,Z -75.923,A -90.000,B 90.000,C 0.000} C_DIS
LIN {X 69.096,Y -40.730,Z -75.934,A -90.000,B 90.000,C 0.000} C_DIS
LIN {X 69.258,Y -40.709,Z -75.977,A -90.000,B 90.000,C 0.000} C_DIS
LIN {X 69.442,Y -40.681,Z -76.029,A -90.000,B 90.000,C 0.000} C_DIS
LIN {X 69.627,Y -40.654,Z -76.089,A -90.000,B 90.000,C 0.000} C_DIS
LIN {X 69.701,Y -40.643,Z -76.119,A -90.000,B 90.000,C 0.000} C_DIS
LIN {X 69.834,Y -40.625,Z -76.182,A -90.000,B 90.000,C 0.000} C_DIS
LIN {X 69.997,Y -40.597,Z -76.263,A -90.000,B 90.000,C 0.000} C_DIS
LIN {X 70.217,Y -40.565,Z -76.390,A -90.000,B 90.000,C 0.000} C_DIS
LIN {X 70.321,Y -40.555,Z -76.462,A -90.000,B 90.000,C 0.000} C_DIS
LIN {X 70.536,Y -40.535,Z -76.620,A -90.000,B 90.000,C 0.000} C_DIS
LIN {X 71.022,Y -40.539,Z -76.953,A -90.000,B 90.000,C 0.000} C_DIS
LIN {X 71.271,Y -40.552,Z -77.152,A -90.000,B 90.000,C 0.000} C_DIS
LIN {X 71.391,Y -40.557,Z -77.267,A -90.000,B 90.000,C 0.000} C_DIS
LIN {X 71.481,Y -40.563,Z -77.351,A -90.000,B 90.000,C 0.000} C_DIS
LIN {X 71.724,Y -40.572,Z -77.586,A -90.000,B 90.000,C 0.000} C_DIS
LIN {X 71.749,Y -40.569,Z -77.602,A -90.000,B 90.000,C 0.000} C_DIS
LIN {X 71.941,Y -40.541,Z -77.728,A -90.000,B 90.000,C 0.000} C_DIS
LIN {X 72.222,Y -40.507,Z -77.934,A -90.000,B 90.000,C 0.000} C_DIS
LIN {X 72.300,Y -40.499,Z -77.994,A -90.000,B 90.000,C 0.000} C_DIS
LIN {X 72.442,Y -40.488,Z -78.117,A -90.000,B 90.000,C 0.000} C_DIS
LIN {X 72.501,Y -40.478,Z -78.153,A -90.000,B 90.000,C 0.000} C_DIS
LIN {X 72.544,Y -40.475,Z -78.179,A -90.000,B 90.000,C 0.000} C_DIS
LIN {X 72.650,Y -40.470,Z -78.248,A -90.000,B 90.000,C 0.000} C_DIS
LIN {X 72.882,Y -40.463,Z -78.409,A -90.000,B 90.000,C 0.000} C_DIS
LIN {X 73.055,Y -40.464,Z -78.542,A -90.000,B 90.000,C 0.000} C_DIS
LIN {X 73.332,Y -40.466,Z -78.783,A -90.000,B 90.000,C 0.000} C_DIS
LIN {X 73.612,Y -40.461,Z -79.032,A -90.000,B 90.000,C 0.000} C_DIS
LIN {X 73.733,Y -40.458,Z -79.141,A -90.000,B 90.000,C 0.000} C_DIS
LIN {X 74.013,Y -40.437,Z -79.379,A -90.000,B 90.000,C 0.000} C_DIS
LIN {X 74.129,Y -40.431,Z -79.484,A -90.000,B 90.000,C 0.000} C_DIS
LIN {X 74.176,Y -40.433,Z -79.524,A -90.000,B 90.000,C 0.000} C_DIS
LIN {X 74.284,Y -40.429,Z -79.594,A -90.000,B 90.000,C 0.000} C_DIS
LIN {X 74.607,Y -40.420,Z -79.819,A -90.000,B 90.000,C 0.000} C_DIS
LIN {X 74.946,Y -40.411,Z -80.058,A -90.000,B 90.000,C 0.000} C_DIS
LIN {X 75.034,Y -40.411,Z -80.124,A -90.000,B 90.000,C 0.000} C_DIS
LIN {X 75.138,Y -40.410,Z -80.211,A -90.000,B 90.000,C 0.000} C_DIS
LIN {X 75.220,Y -40.404,Z -80.269,A -90.000,B 90.000,C 0.000} C_DIS
LIN {X 75.281,Y -40.402,Z -80.316,A -90.000,B 90.000,C 0.000} C_DIS
LIN {X 75.499,Y -40.423,Z -80.469,A -90.000,B 90.000,C 0.000} C_DIS
LIN {X 75.562,Y -40.423,Z -80.502,A -90.000,B 90.000,C 0.000} C_DIS
LIN {X 75.974,Y -40.440,Z -80.689,A -90.000,B 90.000,C 0.000} C_DIS
LIN {X 76.062,Y -40.438,Z -80.720,A -90.000,B 90.000,C 0.000} C_DIS
LIN {X 76.105,Y -40.434,Z -80.728,A -90.000,B 90.000,C 0.000} C_DIS
LIN {X 76.385,Y -40.404,Z -80.786,A -90.000,B 90.000,C 0.000} C_DIS
LIN {X 76.425,Y -40.395,Z -80.787,A -90.000,B 90.000,C 0.000} C_DIS
LIN {X 76.488,Y -40.387,Z -80.785,A -90.000,B 90.000,C 0.000} C_DIS
LIN {X 76.732,Y -40.368,Z -80.773,A -90.000,B 90.000,C 0.000} C_DIS
LIN {X 76.939,Y -40.369,Z -80.754,A -90.000,B 90.000,C 0.000} C_DIS
LIN {X 77.047,Y -40.363,Z -80.732,A -90.000,B 90.000,C 0.000} C_DIS
LIN {X 77.258,Y -40.347,Z -80.681,A -90.000,B 90.000,C 0.000} C_DIS
LIN {X 77.508,Y -40.321,Z -80.624,A -90.000,B 90.000,C 0.000} C_DIS
LIN {X 77.559,Y -40.319,Z -80.611,A -90.000,B 90.000,C 0.000} C_DIS
LIN {X 77.629,Y -40.318,Z -80.593,A -90.000,B 90.000,C 0.000} C_DIS
LIN {X 77.783,Y -40.310,Z -80.558,A -90.000,B 90.000,C 0.000} C_DIS
LIN {X 77.985,Y -40.303,Z -80.517,A -90.000,B 90.000,C 0.000} C_DIS
LIN {X 78.164,Y -40.298,Z -80.463,A -90.000,B 90.000,C 0.000} C_DIS
LIN {X 78.536,Y -40.279,Z -80.355,A -90.000,B 90.000,C 0.000} C_DIS
LIN {X 78.687,Y -40.277,Z -80.308,A -90.000,B 90.000,C 0.000} C_DIS
LIN {X 78.843,Y -40.269,Z -80.249,A -90.000,B 90.000,C 0.000} C_DIS
LIN {X 78.920,Y -40.263,Z -80.222,A -90.000,B 90.000,C 0.000} C_DIS
LIN {X 79.000,Y -40.175,Z -80.057,A -90.000,B 90.000,C 0.000} C_DIS
LIN {X 79.054,Y -40.118,Z -79.954,A -90.000,B 90.000,C 0.000} C_DIS
LIN {X 79.077,Y -40.084,Z -79.894,A -90.000,B 90.000,C 0.000} C_DIS
LIN {X 79.139,Y -39.998,Z -79.739,A -90.000,B 90.000,C 0.000} C_DIS
LIN {X 79.209,Y -39.913,Z -79.581,A -90.000,B 90.000,C 0.000} C_DIS
LIN {X 79.221,Y -39.897,Z -79.532,A -90.000,B 90.000,C 0.000} C_DIS
LIN {X 79.231,Y -39.884,Z -79.412,A -90.000,B 90.000,C 0.000} C_DIS
LIN {X 79.272,Y -39.838,Z -79.030,A -90.000,B 90.000,C 0.000} C_DIS
LIN {X 79.283,Y -39.829,Z -78.944,A -90.000,B 90.000,C 0.000} C_DIS
LIN {X 79.291,Y -39.827,Z -78.700,A -90.000,B 90.000,C 0.000} C_DIS
LIN {X 79.290,Y -39.812,Z -78.501,A -90.000,B 90.000,C 0.000} C_DIS
LIN {X 79.291,Y -39.785,Z -78.109,A -90.000,B 90.000,C 0.000} C_DIS
LIN {X 79.288,Y -39.781,Z -78.014,A -90.000,B 90.000,C 0.000} C_DIS
LIN {X 79.247,Y -39.732,Z -77.379,A -90.000,B 90.000,C 0.000} C_DIS
LIN {X 79.228,Y -39.723,Z -77.193,A -90.000,B 90.000,C 0.000} C_DIS
LIN {X 79.202,Y -39.708,Z -76.777,A -90.000,B 90.000,C 0.000} C_DIS
LIN {X 79.181,Y -39.695,Z -76.479,A -90.000,B 90.000,C 0.000} C_DIS
LIN {X 79.155,Y -39.667,Z -75.962,A -90.000,B 90.000,C 0.000} C_DIS
LIN {X 79.145,Y -39.663,Z -75.832,A -90.000,B 90.000,C 0.000} C_DIS
LIN {X 79.109,Y -39.641,Z -75.497,A -90.000,B 90.000,C 0.000} C_DIS
LIN {X 79.073,Y -39.620,Z -75.124,A -90.000,B 90.000,C 0.000} C_DIS
LIN {X 79.034,Y -39.607,Z -74.798,A -90.000,B 90.000,C 0.000} C_DIS
LIN {X 79.028,Y -39.603,Z -74.729,A -90.000,B 90.000,C 0.000} C_DIS
LIN {X 78.992,Y -39.585,Z -74.174,A -90.000,B 90.000,C 0.000} C_DIS
LIN {X 78.972,Y -39.561,Z -73.668,A -90.000,B 90.000,C 0.000} C_DIS
LIN {X 78.965,Y -39.553,Z -73.479,A -90.000,B 90.000,C 0.000} C_DIS
LIN {X 78.938,Y -39.518,Z -72.878,A -90.000,B 90.000,C 0.000} C_DIS
LIN {X 78.919,Y -39.494,Z -72.422,A -90.000,B 90.000,C 0.000} C_DIS
LIN {X 78.912,Y -39.485,Z -72.167,A -90.000,B 90.000,C 0.000} C_DIS
LIN {X 78.915,Y -39.468,Z -71.754,A -90.000,B 90.000,C 0.000} C_DIS
LIN {X 78.931,Y -39.453,Z -71.245,A -90.000,B 90.000,C 0.000} C_DIS
LIN {X 78.945,Y -39.446,Z -71.088,A -90.000,B 90.000,C 0.000} C_DIS
LIN {X 79.014,Y -39.419,Z -70.323,A -90.000,B 90.000,C 0.000} C_DIS
LIN {X 79.094,Y -39.395,Z -69.886,A -90.000,B 90.000,C 0.000} C_DIS
LIN {X 79.153,Y -39.380,Z -69.585,A -90.000,B 90.000,C 0.000} C_DIS
LIN {X 79.260,Y -39.360,Z -69.036,A -90.000,B 90.000,C 0.000} C_DIS
LIN {X 79.351,Y -39.348,Z -68.620,A -90.000,B 90.000,C 0.000} C_DIS
LIN {X 79.498,Y -39.334,Z -68.166,A -90.000,B 90.000,C 0.000} C_DIS
LIN {X 79.676,Y -39.324,Z -67.623,A -90.000,B 90.000,C 0.000} C_DIS
LIN {X 79.789,Y -39.318,Z -67.300,A -90.000,B 90.000,C 0.000} C_DIS
LIN {X 79.868,Y -39.316,Z -67.089,A -90.000,B 90.000,C 0.000} C_DIS
LIN {X 79.923,Y -39.315,Z -66.958,A -90.000,B 90.000,C 0.000} C_DIS
LIN {X 80.093,Y -39.311,Z -66.571,A -90.000,B 90.000,C 0.000} C_DIS
LIN {X 80.394,Y -39.309,Z -65.888,A -90.000,B 90.000,C 0.000} C_DIS
LIN {X 80.639,Y -39.309,Z -65.345,A -90.000,B 90.000,C 0.000} C_DIS
LIN {X 80.673,Y -39.309,Z -65.279,A -90.000,B 90.000,C 0.000} C_DIS
LIN {X 81.101,Y -39.317,Z -64.454,A -90.000,B 90.000,C 0.000} C_DIS
LIN {X 81.114,Y -39.320,Z -64.429,A -90.000,B 90.000,C 0.000} C_DIS
LIN {X 81.298,Y -39.318,Z -64.075,A -90.000,B 90.000,C 0.000} C_DIS
LIN {X 81.438,Y -39.308,Z -63.804,A -90.000,B 90.000,C 0.000} C_DIS
LIN {X 81.438,Y -60.000,Z -63.804,A -90.000,B 90.000,C 0.000} C_DIS
LIN {X 89.672,Y -60.000,Z -53.967,A -90.000,B 90.000,C 0.000} C_DIS
LIN {X 89.672,Y -39.308,Z -53.967,A -90.000,B 90.000,C 0.000} C_DIS
LIN {X 89.730,Y -39.308,Z -53.914,A -90.000,B 90.000,C 0.000} C_DIS
LIN {X 89.730,Y -60.000,Z -53.914,A -90.000,B 90.000,C 0.000} C_DIS
LIN {X 97.702,Y -60.000,Z -46.864,A -90.000,B 90.000,C 0.000} C_DIS
LIN {X 97.702,Y -39.308,Z -46.864,A -90.000,B 90.000,C 0.000} C_DIS
LIN {X 97.877,Y -39.308,Z -46.679,A -90.000,B 90.000,C 0.000} C_DIS
LIN {X 98.223,Y -44.514,Z -46.315,A -90.000,B 90.000,C 0.000} C_DIS
LIN {X 98.483,Y -44.409,Z -46.043,A -90.000,B 90.000,C 0.000} C_DIS
LIN {X 98.670,Y -44.352,Z -45.848,A -90.000,B 90.000,C 0.000} C_DIS
LIN {X 98.797,Y -44.328,Z -45.718,A -90.000,B 90.000,C 0.000} C_DIS
LIN {X 98.874,Y -44.327,Z -45.640,A -90.000,B 90.000,C 0.000} C_DIS
LIN {X 98.898,Y -44.332,Z -45.616,A -90.000,B 90.000,C 0.000} C_DIS
LIN {X 98.914,Y -44.339,Z -45.600,A -90.000,B 90.000,C 0.000} C_DIS
LIN {X 98.930,Y -44.355,Z -45.586,A -90.000,B 90.000,C 0.000} C_DIS
LIN {X 98.933,Y -44.368,Z -45.585,A -90.000,B 90.000,C 0.000} C_DIS
LIN {X 99.058,Y -44.166,Z -45.441,A -90.000,B 90.000,C 0.000} C_DIS
LIN {X 99.357,Y -43.911,Z -45.104,A -90.000,B 90.000,C 0.000} C_DIS
LIN {X 99.608,Y -43.722,Z -44.823,A -90.000,B 90.000,C 0.000} C_DIS
LIN {X 99.943,Y -39.308,Z -44.450,A -90.000,B 90.000,C 0.000} C_DIS
LIN {X 100.003,Y -39.310,Z -44.383,A -90.000,B 90.000,C 0.000} C_DIS
LIN {X 100.056,Y -39.308,Z -44.323,A -90.000,B 90.000,C 0.000} C_DIS
LIN {X 100.361,Y -43.219,Z -43.983,A -90.000,B 90.000,C 0.000} C_DIS
LIN {X 100.518,Y -43.132,Z -43.809,A -90.000,B 90.000,C 0.000} C_DIS
LIN {X 100.575,Y -43.094,Z -43.744,A -90.000,B 90.000,C 0.000} C_DIS
LIN {X 100.582,Y -43.085,Z -43.736,A -90.000,B 90.000,C 0.000} C_DIS
LIN {X 100.583,Y -43.066,Z -43.733,A -90.000,B 90.000,C 0.000} C_DIS
LIN {X 100.590,Y -43.049,Z -43.724,A -90.000,B 90.000,C 0.000} C_DIS
LIN {X 100.647,Y -42.983,Z -43.659,A -90.000,B 90.000,C 0.000} C_DIS
LIN {X 100.802,Y -42.848,Z -43.483,A -90.000,B 90.000,C 0.000} C_DIS
LIN {X 101.104,Y -39.308,Z -43.141,A -90.000,B 90.000,C 0.000} C_DIS
LIN {X 101.165,Y -39.308,Z -43.073,A -90.000,B 90.000,C 0.000} C_DIS
LIN {X 101.306,Y -42.474,Z -42.913,A -90.000,B 90.000,C 0.000} C_DIS
LIN {X 101.326,Y -42.463,Z -42.891,A -90.000,B 90.000,C 0.000} C_DIS
LIN {X 101.329,Y -42.473,Z -42.888,A -90.000,B 90.000,C 0.000} C_DIS
LIN {X 101.347,Y -42.474,Z -42.869,A -90.000,B 90.000,C 0.000} C_DIS
LIN {X 101.490,Y -39.308,Z -42.711,A -90.000,B 90.000,C 0.000} C_DIS
LIN {X 101.527,Y -39.308,Z -42.670,A -90.000,B 90.000,C 0.000} C_DIS
LIN {X 101.953,Y -41.785,Z -42.197,A -90.000,B 90.000,C 0.000} C_DIS
LIN {X 102.007,Y -41.721,Z -42.138,A -90.000,B 90.000,C 0.000} C_DIS
LIN {X 102.014,Y -41.732,Z -42.131,A -90.000,B 90.000,C 0.000} C_DIS
LIN {X 102.016,Y -41.778,Z -42.130,A -90.000,B 90.000,C 0.000} C_DIS
LIN {X 102.023,Y -41.796,Z -42.123,A -90.000,B 90.000,C 0.000} C_DIS
LIN {X 102.078,Y -41.787,Z -42.065,A -90.000,B 90.000,C 0.000} C_DIS
LIN {X 102.224,Y -41.679,Z -41.906,A -90.000,B 90.000,C 0.000} C_DIS
LIN {X 102.508,Y -39.308,Z -41.596,A -90.000,B 90.000,C 0.000} C_DIS
LIN {X 102.577,Y -39.308,Z -41.520,A -90.000,B 90.000,C 0.000} C_DIS
LIN {X 102.653,Y -41.243,Z -41.437,A -90.000,B 90.000,C 0.000} C_DIS
LIN {X 102.663,Y -41.229,Z -41.426,A -90.000,B 90.000,C 0.000} C_DIS
LIN {X 102.676,Y -41.250,Z -41.414,A -90.000,B 90.000,C 0.000} C_DIS
LIN {X 102.753,Y -39.308,Z -41.331,A -90.000,B 90.000,C 0.000} C_DIS
LIN {X 103.579,Y -39.309,Z -40.452,A -90.000,B 90.000,C 0.000} C_DIS
LIN {X 104.447,Y -39.313,Z -39.580,A -90.000,B 90.000,C 0.000} C_DIS
LIN {X 104.780,Y -39.317,Z -39.269,A -90.000,B 90.000,C 0.000} C_DIS
LIN {X 105.187,Y -39.325,Z -38.863,A -90.000,B 90.000,C 0.000} C_DIS
LIN {X 105.542,Y -39.332,Z -38.542,A -90.000,B 90.000,C 0.000} C_DIS
LIN {X 105.806,Y -39.339,Z -38.316,A -90.000,B 90.000,C 0.000} C_DIS
LIN {X 106.173,Y -39.352,Z -38.002,A -90.000,B 90.000,C 0.000} C_DIS
LIN {X 106.715,Y -39.370,Z -37.601,A -90.000,B 90.000,C 0.000} C_DIS
LIN {X 106.864,Y -39.375,Z -37.496,A -90.000,B 90.000,C 0.000} C_DIS
LIN {X 107.009,Y -39.378,Z -37.399,A -90.000,B 90.000,C 0.000} C_DIS
LIN {X 107.123,Y -39.382,Z -37.325,A -90.000,B 90.000,C 0.000} C_DIS
LIN {X 107.483,Y -39.396,Z -37.113,A -90.000,B 90.000,C 0.000} C_DIS
LIN {X 107.945,Y -39.407,Z -36.871,A -90.000,B 90.000,C 0.000} C_DIS
LIN {X 108.132,Y -39.412,Z -36.782,A -90.000,B 90.000,C 0.000} C_DIS
LIN {X 108.381,Y -39.423,Z -36.667,A -90.000,B 90.000,C 0.000} C_DIS
LIN {X 108.815,Y -39.427,Z -36.512,A -90.000,B 90.000,C 0.000} C_DIS
LIN {X 109.214,Y -39.441,Z -36.375,A -90.000,B 90.000,C 0.000} C_DIS
LIN {X 109.279,Y -39.441,Z -36.359,A -90.000,B 90.000,C 0.000} C_DIS
LIN {X 109.355,Y -39.442,Z -36.341,A -90.000,B 90.000,C 0.000} C_DIS
LIN {X 109.684,Y -39.454,Z -36.262,A -90.000,B 90.000,C 0.000} C_DIS
LIN {X 110.142,Y -39.456,Z -36.198,A -90.000,B 90.000,C 0.000} C_DIS
LIN {X 110.495,Y -39.466,Z -36.151,A -90.000,B 90.000,C 0.000} C_DIS
LIN {X 110.674,Y -39.468,Z -36.143,A -90.000,B 90.000,C 0.000} C_DIS
LIN {X 110.974,Y -39.476,Z -36.135,A -90.000,B 90.000,C 0.000} C_DIS
LIN {X 111.151,Y -39.476,Z -36.143,A -90.000,B 90.000,C 0.000} C_DIS
LIN {X 111.479,Y -39.477,Z -36.159,A -90.000,B 90.000,C 0.000} C_DIS
LIN {X 111.736,Y -39.485,Z -36.179,A -90.000,B 90.000,C 0.000} C_DIS
LIN {X 111.888,Y -39.486,Z -36.203,A -90.000,B 90.000,C 0.000} C_DIS
LIN {X 112.208,Y -39.492,Z -36.259,A -90.000,B 90.000,C 0.000} C_DIS
LIN {X 112.433,Y -39.494,Z -36.313,A -90.000,B 90.000,C 0.000} C_DIS
LIN {X 112.726,Y -39.495,Z -36.391,A -90.000,B 90.000,C 0.000} C_DIS
LIN {X 112.893,Y -39.501,Z -36.439,A -90.000,B 90.000,C 0.000} C_DIS
LIN {X 113.150,Y -39.504,Z -36.536,A -90.000,B 90.000,C 0.000} C_DIS
LIN {X 113.317,Y -39.507,Z -36.601,A -90.000,B 90.000,C 0.000} C_DIS
LIN {X 113.435,Y -39.514,Z -36.648,A -90.000,B 90.000,C 0.000} C_DIS
LIN {X 113.508,Y -39.516,Z -36.683,A -90.000,B 90.000,C 0.000} C_DIS
LIN {X 113.980,Y -39.524,Z -36.922,A -90.000,B 90.000,C 0.000} C_DIS
LIN {X 114.171,Y -39.534,Z -37.024,A -90.000,B 90.000,C 0.000} C_DIS
LIN {X 114.257,Y -39.537,Z -37.077,A -90.000,B 90.000,C 0.000} C_DIS
LIN {X 114.310,Y -39.540,Z -37.107,A -90.000,B 90.000,C 0.000} C_DIS
LIN {X 114.389,Y -39.542,Z -37.157,A -90.000,B 90.000,C 0.000} C_DIS
LIN {X 114.451,Y -39.545,Z -37.197,A -90.000,B 90.000,C 0.000} C_DIS
LIN {X 114.696,Y -39.565,Z -37.358,A -90.000,B 90.000,C 0.000} C_DIS
LIN {X 115.057,Y -39.580,Z -37.647,A -90.000,B 90.000,C 0.000} C_DIS
LIN {X 115.216,Y -39.583,Z -37.803,A -90.000,B 90.000,C 0.000} C_DIS
LIN {X 115.388,Y -39.590,Z -37.974,A -90.000,B 90.000,C 0.000} C_DIS
LIN {X 115.446,Y -39.589,Z -38.042,A -90.000,B 90.000,C 0.000} C_DIS
LIN {X 115.686,Y -39.599,Z -38.336,A -90.000,B 90.000,C 0.000} C_DIS
LIN {X 115.759,Y -39.599,Z -38.435,A -90.000,B 90.000,C 0.000} C_DIS
LIN {X 115.883,Y -39.605,Z -38.599,A -90.000,B 90.000,C 0.000} C_DIS
LIN {X 115.935,Y -39.605,Z -38.676,A -90.000,B 90.000,C 0.000} C_DIS
LIN {X 116.130,Y -39.614,Z -38.977,A -90.000,B 90.000,C 0.000} C_DIS
LIN {X 116.209,Y -39.613,Z -39.121,A -90.000,B 90.000,C 0.000} C_DIS
LIN {X 116.353,Y -39.617,Z -39.401,A -90.000,B 90.000,C 0.000} C_DIS
LIN {X 116.405,Y -39.615,Z -39.525,A -90.000,B 90.000,C 0.000} C_DIS
LIN {X 116.489,Y -39.617,Z -39.707,A -90.000,B 90.000,C 0.000} C_DIS
LIN {X 116.558,Y -39.615,Z -39.879,A -90.000,B 90.000,C 0.000} C_DIS
LIN {X 116.658,Y -39.621,Z -40.141,A -90.000,B 90.000,C 0.000} C_DIS
LIN {X 116.676,Y -39.619,Z -40.203,A -90.000,B 90.000,C 0.000} C_DIS
LIN {X 116.743,Y -39.618,Z -40.424,A -90.000,B 90.000,C 0.000} C_DIS
LIN {X 116.803,Y -39.615,Z -40.641,A -90.000,B 90.000,C 0.000} C_DIS
LIN {X 116.833,Y -39.616,Z -40.752,A -90.000,B 90.000,C 0.000} C_DIS
LIN {X 116.866,Y -39.622,Z -40.881,A -90.000,B 90.000,C 0.000} C_DIS
LIN {X 116.943,Y -39.617,Z -41.343,A -90.000,B 90.000,C 0.000} C_DIS
LIN {X 116.956,Y -39.615,Z -41.446,A -90.000,B 90.000,C 0.000} C_DIS
LIN {X 116.976,Y -39.618,Z -41.616,A -90.000,B 90.000,C 0.000} C_DIS
LIN {X 116.995,Y -39.617,Z -41.966,A -90.000,B 90.000,C 0.000} C_DIS
LIN {X 117.000,Y -39.619,Z -42.082,A -90.000,B 90.000,C 0.000} C_DIS
LIN {X 116.997,Y -39.616,Z -42.197,A -90.000,B 90.000,C 0.000} C_DIS
LIN {X 116.988,Y -39.613,Z -42.438,A -90.000,B 90.000,C 0.000} C_DIS
LIN {X 116.970,Y -39.614,Z -42.668,A -90.000,B 90.000,C 0.000} C_DIS
LIN {X 116.948,Y -39.611,Z -42.852,A -90.000,B 90.000,C 0.000} C_DIS
LIN {X 116.931,Y -39.611,Z -42.973,A -90.000,B 90.000,C 0.000} C_DIS
LIN {X 116.909,Y -39.617,Z -43.123,A -90.000,B 90.000,C 0.000} C_DIS
LIN {X 116.803,Y -39.612,Z -43.579,A -90.000,B 90.000,C 0.000} C_DIS
LIN {X 116.779,Y -39.610,Z -43.667,A -90.000,B 90.000,C 0.000} C_DIS
LIN {X 116.729,Y -39.614,Z -43.840,A -90.000,B 90.000,C 0.000} C_DIS
LIN {X 116.646,Y -39.613,Z -44.084,A -90.000,B 90.000,C 0.000} C_DIS
LIN {X 116.599,Y -39.616,Z -44.226,A -90.000,B 90.000,C 0.000} C_DIS
LIN {X 116.540,Y -39.625,Z -44.399,A -90.000,B 90.000,C 0.000} C_DIS
LIN {X 116.402,Y -39.658,Z -44.814,A -90.000,B 90.000,C 0.000} C_DIS
LIN {X 116.344,Y -39.673,Z -44.979,A -90.000,B 90.000,C 0.000} C_DIS
LIN {X 116.204,Y -39.718,Z -45.362,A -90.000,B 90.000,C 0.000} C_DIS
LIN {X 116.178,Y -39.721,Z -45.442,A -90.000,B 90.000,C 0.000} C_DIS
LIN {X 116.150,Y -39.719,Z -45.532,A -90.000,B 90.000,C 0.000} C_DIS
LIN {X 116.070,Y -39.711,Z -45.806,A -90.000,B 90.000,C 0.000} C_DIS
LIN {X 115.903,Y -39.682,Z -46.354,A -90.000,B 90.000,C 0.000} C_DIS
LIN {X 115.837,Y -39.669,Z -46.563,A -90.000,B 90.000,C 0.000} C_DIS
LIN {X 115.613,Y -39.630,Z -47.221,A -90.000,B 90.000,C 0.000} C_DIS
LIN {X 115.502,Y -39.617,Z -47.539,A -90.000,B 90.000,C 0.000} C_DIS
LIN {X 115.438,Y -39.608,Z -47.713,A -90.000,B 90.000,C 0.000} C_DIS
LIN {X 115.181,Y -39.563,Z -48.352,A -90.000,B 90.000,C 0.000} C_DIS
LIN {X 115.071,Y -39.550,Z -48.616,A -90.000,B 90.000,C 0.000} C_DIS
LIN {X 115.032,Y -39.547,Z -48.711,A -90.000,B 90.000,C 0.000} C_DIS
LIN {X 114.971,Y -39.540,Z -48.848,A -90.000,B 90.000,C 0.000} C_DIS
LIN {X 114.749,Y -39.514,Z -49.332,A -90.000,B 90.000,C 0.000} C_DIS
LIN {X 114.475,Y -39.486,Z -49.926,A -90.000,B 90.000,C 0.000} C_DIS
LIN {X 114.283,Y -39.477,Z -50.330,A -90.000,B 90.000,C 0.000} C_DIS
LIN {X 113.949,Y -39.460,Z -51.017,A -90.000,B 90.000,C 0.000} C_DIS
LIN {X 113.718,Y -39.449,Z -51.487,A -90.000,B 90.000,C 0.000} C_DIS
LIN {X 113.133,Y -39.431,Z -52.708,A -90.000,B 90.000,C 0.000} C_DIS
LIN {X 112.451,Y -39.431,Z -54.211,A -90.000,B 90.000,C 0.000} C_DIS
LIN {X 111.777,Y -39.432,Z -55.808,A -90.000,B 90.000,C 0.000} C_DIS
LIN {X 111.586,Y -39.433,Z -56.303,A -90.000,B 90.000,C 0.000} C_DIS
LIN {X 111.161,Y -39.434,Z -57.388,A -90.000,B 90.000,C 0.000} C_DIS
LIN {X 111.106,Y -39.436,Z -57.540,A -90.000,B 90.000,C 0.000} C_DIS
LIN {X 110.612,Y -39.439,Z -58.899,A -90.000,B 90.000,C 0.000} C_DIS
LIN {X 110.543,Y -39.441,Z -59.103,A -90.000,B 90.000,C 0.000} C_DIS
LIN {X 109.945,Y -39.444,Z -60.876,A -90.000,B 90.000,C 0.000} C_DIS
LIN {X 109.425,Y -39.447,Z -62.439,A -90.000,B 90.000,C 0.000} C_DIS
LIN {X 109.199,Y -39.448,Z -63.116,A -90.000,B 90.000,C 0.000} C_DIS
LIN {X 108.478,Y -39.456,Z -65.222,A -90.000,B 90.000,C 0.000} C_DIS
LIN {X 108.289,Y -39.455,Z -65.741,A -90.000,B 90.000,C 0.000} C_DIS
LIN {X 107.471,Y -39.466,Z -67.953,A -90.000,B 90.000,C 0.000} C_DIS
LIN {X 106.788,Y -39.479,Z -69.618,A -90.000,B 90.000,C 0.000} C_DIS
LIN {X 106.505,Y -39.484,Z -70.299,A -90.000,B 90.000,C 0.000} C_DIS
LIN {X 106.307,Y -39.484,Z -70.742,A -90.000,B 90.000,C 0.000} C_DIS
LIN {X 105.683,Y -39.495,Z -72.117,A -90.000,B 90.000,C 0.000} C_DIS
LIN {X 105.421,Y -39.503,Z -72.691,A -90.000,B 90.000,C 0.000} C_DIS
LIN {X 105.216,Y -39.504,Z -73.111,A -90.000,B 90.000,C 0.000} C_DIS
LIN {X 104.841,Y -39.512,Z -73.870,A -90.000,B 90.000,C 0.000} C_DIS
LIN {X 104.073,Y -39.539,Z -75.403,A -90.000,B 90.000,C 0.000} C_DIS
LIN {X 103.797,Y -39.543,Z -75.908,A -90.000,B 90.000,C 0.000} C_DIS
LIN {X 103.369,Y -39.563,Z -76.682,A -90.000,B 90.000,C 0.000} C_DIS
LIN {X 102.858,Y -39.576,Z -77.567,A -90.000,B 90.000,C 0.000} C_DIS
LIN {X 102.558,Y -39.574,Z -78.045,A -90.000,B 90.000,C 0.000} C_DIS
LIN {X 102.070,Y -39.598,Z -78.794,A -90.000,B 90.000,C 0.000} C_DIS
LIN {X 101.607,Y -39.615,Z -79.482,A -90.000,B 90.000,C 0.000} C_DIS
LIN {X 101.388,Y -39.615,Z -79.784,A -90.000,B 90.000,C 0.000} C_DIS
LIN {X 101.084,Y -39.626,Z -80.194,A -90.000,B 90.000,C 0.000} C_DIS
LIN {X 100.546,Y -39.655,Z -80.911,A -90.000,B 90.000,C 0.000} C_DIS
LIN {X 100.163,Y -39.676,Z -81.418,A -90.000,B 90.000,C 0.000} C_DIS
LIN {X 99.889,Y -39.684,Z -81.761,A -90.000,B 90.000,C 0.000} C_DIS
LIN {X 99.203,Y -39.730,Z -82.604,A -90.000,B 90.000,C 0.000} C_DIS
LIN {X 99.037,Y -39.737,Z -82.799,A -90.000,B 90.000,C 0.000} C_DIS
LIN {X 98.699,Y -39.744,Z -83.181,A -90.000,B 90.000,C 0.000} C_DIS
LIN {X 98.346,Y -39.764,Z -83.568,A -90.000,B 90.000,C 0.000} C_DIS
LIN {X 98.203,Y -39.775,Z -83.722,A -90.000,B 90.000,C 0.000} C_DIS
LIN {X 97.945,Y -39.784,Z -83.982,A -90.000,B 90.000,C 0.000} C_DIS
LIN {X 97.724,Y -39.789,Z -84.199,A -90.000,B 90.000,C 0.000} C_DIS
LIN {X 97.526,Y -39.793,Z -84.391,A -90.000,B 90.000,C 0.000} C_DIS
LIN {X 97.087,Y -39.821,Z -84.794,A -90.000,B 90.000,C 0.000} C_DIS
LIN {X 96.582,Y -39.868,Z -85.226,A -90.000,B 90.000,C 0.000} C_DIS
LIN {X 96.308,Y -39.892,Z -85.453,A -90.000,B 90.000,C 0.000} C_DIS
LIN {X 95.741,Y -39.955,Z -85.905,A -90.000,B 90.000,C 0.000} C_DIS
LIN {X 95.473,Y -39.990,Z -86.114,A -90.000,B 90.000,C 0.000} C_DIS
LIN {X 94.646,Y -40.050,Z -86.699,A -90.000,B 90.000,C 0.000} C_DIS
LIN {X 94.494,Y -40.052,Z -86.796,A -90.000,B 90.000,C 0.000} C_DIS
LIN {X 94.137,Y -40.070,Z -87.006,A -90.000,B 90.000,C 0.000} C_DIS
LIN {X 93.573,Y -40.109,Z -87.331,A -90.000,B 90.000,C 0.000} C_DIS
LIN {X 93.506,Y -40.114,Z -87.368,A -90.000,B 90.000,C 0.000} C_DIS
LIN {X 93.108,Y -40.153,Z -87.580,A -90.000,B 90.000,C 0.000} C_DIS
LIN {X 93.040,Y -40.165,Z -87.620,A -90.000,B 90.000,C 0.000} C_DIS
LIN {X 92.703,Y -40.207,Z -87.843,A -90.000,B 90.000,C 0.000} C_DIS
LIN {X 92.542,Y -40.218,Z -87.941,A -90.000,B 90.000,C 0.000} C_DIS
LIN {X 92.382,Y -40.243,Z -88.049,A -90.000,B 90.000,C 0.000} C_DIS
LIN {X 92.185,Y -40.271,Z -88.177,A -90.000,B 90.000,C 0.000} C_DIS
LIN {X 92.158,Y -40.279,Z -88.196,A -90.000,B 90.000,C 0.000} C_DIS
LIN {X 91.943,Y -40.327,Z -88.379,A -90.000,B 90.000,C 0.000} C_DIS
LIN {X 91.887,Y -40.346,Z -88.425,A -90.000,B 90.000,C 0.000} C_DIS
LIN {X 91.818,Y -40.339,Z -88.592,A -90.000,B 90.000,C 0.000} C_DIS
LIN {X 91.784,Y -40.337,Z -88.679,A -90.000,B 90.000,C 0.000} C_DIS
LIN {X 91.750,Y -40.327,Z -88.820,A -90.000,B 90.000,C 0.000} C_DIS
LIN {X 91.626,Y -40.309,Z -89.379,A -90.000,B 90.000,C 0.000} C_DIS
LIN {X 91.608,Y -40.311,Z -89.474,A -90.000,B 90.000,C 0.000} C_DIS
LIN {X 91.508,Y -40.288,Z -90.434,A -90.000,B 90.000,C 0.000} C_DIS
LIN {X 91.482,Y -40.278,Z -90.654,A -90.000,B 90.000,C 0.000} C_DIS
LIN {X 91.460,Y -40.261,Z -90.904,A -90.000,B 90.000,C 0.000} C_DIS
LIN {X 91.366,Y -40.235,Z -92.289,A -90.000,B 90.000,C 0.000} C_DIS
LIN {X 91.223,Y -40.210,Z -94.052,A -90.000,B 90.000,C 0.000} C_DIS
LIN {X 91.201,Y -40.210,Z -94.278,A -90.000,B 90.000,C 0.000} C_DIS
LIN {X 91.182,Y -40.205,Z -94.442,A -90.000,B 90.000,C 0.000} C_DIS
LIN {X 91.170,Y -40.204,Z -94.534,A -90.000,B 90.000,C 0.000} C_DIS
LIN {X 90.946,Y -40.201,Z -95.972,A -90.000,B 90.000,C 0.000} C_DIS
LIN {X 90.925,Y -40.202,Z -96.089,A -90.000,B 90.000,C 0.000} C_DIS
LIN {X 90.822,Y -40.193,Z -96.483,A -90.000,B 90.000,C 0.000} C_DIS
LIN {X 90.767,Y -40.193,Z -96.654,A -90.000,B 90.000,C 0.000} C_DIS
LIN {X 90.622,Y -40.201,Z -97.048,A -90.000,B 90.000,C 0.000} C_DIS
LIN {X 90.451,Y -40.214,Z -97.516,A -90.000,B 90.000,C 0.000} C_DIS
LIN {X 90.310,Y -40.206,Z -97.865,A -90.000,B 90.000,C 0.000} C_DIS
LIN {X 90.237,Y -40.195,Z -98.026,A -90.000,B 90.000,C 0.000} C_DIS
LIN {X 90.182,Y -40.189,Z -98.139,A -90.000,B 90.000,C 0.000} C_DIS
LIN {X 90.117,Y -40.188,Z -98.258,A -90.000,B 90.000,C 0.000} C_DIS
LIN {X 89.955,Y -40.190,Z -98.541,A -90.000,B 90.000,C 0.000} C_DIS
LIN {X 89.886,Y -40.194,Z -98.656,A -90.000,B 90.000,C 0.000} C_DIS
LIN {X 89.657,Y -40.207,Z -99.001,A -90.000,B 90.000,C 0.000} C_DIS
LIN {X 89.362,Y -40.195,Z -99.417,A -90.000,B 90.000,C 0.000} C_DIS
LIN {X 89.300,Y -40.195,Z -99.501,A -90.000,B 90.000,C 0.000} C_DIS
LIN {X 89.085,Y -40.198,Z -99.778,A -90.000,B 90.000,C 0.000} C_DIS
LIN {X 88.982,Y -40.201,Z -99.900,A -90.000,B 90.000,C 0.000} C_DIS
LIN {X 88.850,Y -40.210,Z -100.046,A -90.000,B 90.000,C 0.000} C_DIS
LIN {X 88.380,Y -40.210,Z -100.550,A -90.000,B 90.000,C 0.000} C_DIS
LIN {X 88.297,Y -40.216,Z -100.641,A -90.000,B 90.000,C 0.000} C_DIS
LIN {X 88.050,Y -40.239,Z -100.899,A -90.000,B 90.000,C 0.000} C_DIS
LIN {X 87.959,Y -40.250,Z -100.989,A -90.000,B 90.000,C 0.000} C_DIS
LIN {X 87.735,Y -40.280,Z -101.197,A -90.000,B 90.000,C 0.000} C_DIS
LIN {X 87.611,Y -40.306,Z -101.319,A -90.000,B 90.000,C 0.000} C_DIS
LIN {X 87.168,Y -40.373,Z -101.837,A -90.000,B 90.000,C 0.000} C_DIS
LIN {X 87.049,Y -40.381,Z -102.007,A -90.000,B 90.000,C 0.000} C_DIS
LIN {X 86.743,Y -40.436,Z -102.473,A -90.000,B 90.000,C 0.000} C_DIS
LIN {X 86.570,Y -40.448,Z -102.814,A -90.000,B 90.000,C 0.000} C_DIS
LIN {X 86.470,Y -40.474,Z -103.028,A -90.000,B 90.000,C 0.000} C_DIS
LIN {X 86.393,Y -40.481,Z -103.291,A -90.000,B 90.000,C 0.000} C_DIS
LIN {X 86.388,Y -40.469,Z -103.402,A -90.000,B 90.000,C 0.000} C_DIS
LIN {X 86.390,Y -40.472,Z -103.515,A -90.000,B 90.000,C 0.000} C_DIS
LIN {X 86.446,Y -40.455,Z -103.994,A -90.000,B 90.000,C 0.000} C_DIS
LIN {X 86.459,Y -40.458,Z -104.083,A -90.000,B 90.000,C 0.000} C_DIS
LIN {X 86.515,Y -40.454,Z -104.324,A -90.000,B 90.000,C 0.000} C_DIS
LIN {X 86.553,Y -40.456,Z -104.528,A -90.000,B 90.000,C 0.000} C_DIS
LIN {X 86.612,Y -40.480,Z -105.060,A -90.000,B 90.000,C 0.000} C_DIS
LIN {X 86.636,Y -40.488,Z -105.292,A -90.000,B 90.000,C 0.000} C_DIS
LIN {X 86.745,Y -40.471,Z -105.825,A -90.000,B 90.000,C 0.000} C_DIS
LIN {X 86.775,Y -40.469,Z -105.990,A -90.000,B 90.000,C 0.000} C_DIS
LIN {X 86.786,Y -40.471,Z -106.084,A -90.000,B 90.000,C 0.000} C_DIS
LIN {X 86.815,Y -40.479,Z -106.362,A -90.000,B 90.000,C 0.000} C_DIS
LIN {X 86.819,Y -40.479,Z -106.425,A -90.000,B 90.000,C 0.000} C_DIS
LIN {X 86.823,Y -40.482,Z -106.527,A -90.000,B 90.000,C 0.000} C_DIS
LIN {X 86.821,Y -40.491,Z -106.728,A -90.000,B 90.000,C 0.000} C_DIS
LIN {X 86.817,Y -40.497,Z -106.819,A -90.000,B 90.000,C 0.000} C_DIS
LIN {X 86.794,Y -40.514,Z -107.159,A -90.000,B 90.000,C 0.000} C_DIS
LIN {X 86.821,Y -40.505,Z -108.059,A -90.000,B 90.000,C 0.000} C_DIS
LIN {X 86.821,Y -40.506,Z -108.196,A -90.000,B 90.000,C 0.000} C_DIS
LIN {X 86.817,Y -40.509,Z -108.326,A -90.000,B 90.000,C 0.000} C_DIS
LIN {X 86.800,Y -40.509,Z -108.509,A -90.000,B 90.000,C 0.000} C_DIS
LIN {X 86.780,Y -40.513,Z -108.644,A -90.000,B 90.000,C 0.000} C_DIS
LIN {X 86.747,Y -40.514,Z -108.838,A -90.000,B 90.000,C 0.000} C_DIS
LIN {X 86.707,Y -40.518,Z -109.024,A -90.000,B 90.000,C 0.000} C_DIS
LIN {X 86.678,Y -40.524,Z -109.126,A -90.000,B 90.000,C 0.000} C_DIS
LIN {X 86.488,Y -40.569,Z -109.734,A -90.000,B 90.000,C 0.000} C_DIS
LIN {X 86.353,Y -40.587,Z -110.312,A -90.000,B 90.000,C 0.000} C_DIS
LIN {X 86.284,Y -40.604,Z -110.621,A -90.000,B 90.000,C 0.000} C_DIS
LIN {X 86.205,Y -40.603,Z -110.941,A -90.000,B 90.000,C 0.000} C_DIS
LIN {X 86.149,Y -40.608,Z -111.130,A -90.000,B 90.000,C 0.000} C_DIS
LIN {X 86.058,Y -40.620,Z -111.397,A -90.000,B 90.000,C 0.000} C_DIS
LIN {X 86.012,Y -40.628,Z -111.518,A -90.000,B 90.000,C 0.000} C_DIS
LIN {X 85.861,Y -40.658,Z -111.887,A -90.000,B 90.000,C 0.000} C_DIS
LIN {X 85.791,Y -40.669,Z -112.055,A -90.000,B 90.000,C 0.000} C_DIS
LIN {X 85.526,Y -40.702,Z -112.683,A -90.000,B 90.000,C 0.000} C_DIS
LIN {X 85.273,Y -40.723,Z -113.385,A -90.000,B 90.000,C 0.000} C_DIS
LIN {X 85.197,Y -40.724,Z -113.590,A -90.000,B 90.000,C 0.000} C_DIS
LIN {X 85.137,Y -40.725,Z -113.747,A -90.000,B 90.000,C 0.000} C_DIS
LIN {X 84.486,Y -40.745,Z -115.290,A -90.000,B 90.000,C 0.000} C_DIS
LIN {X 84.456,Y -40.747,Z -115.363,A -90.000,B 90.000,C 0.000} C_DIS
LIN {X 84.300,Y -40.758,Z -115.779,A -90.000,B 90.000,C 0.000} C_DIS
LIN {X 83.828,Y -40.762,Z -117.392,A -90.000,B 90.000,C 0.000} C_DIS
LIN {X 83.763,Y -40.776,Z -117.630,A -90.000,B 90.000,C 0.000} C_DIS
LIN {X 83.751,Y -40.760,Z -118.814,A -90.000,B 90.000,C 0.000} C_DIS
LIN {X 83.748,Y -40.760,Z -119.178,A -90.000,B 90.000,C 0.000} C_DIS
LIN {X 83.790,Y -40.747,Z -119.417,A -90.000,B 90.000,C 0.000} C_DIS
LIN {X 84.016,Y -40.717,Z -120.644,A -90.000,B 90.000,C 0.000} C_DIS
LIN {X 84.073,Y -40.717,Z -120.948,A -90.000,B 90.000,C 0.000} C_DIS
LIN {X 84.190,Y -40.705,Z -121.376,A -90.000,B 90.000,C 0.000} C_DIS
LIN {X 84.474,Y -40.673,Z -122.423,A -90.000,B 90.000,C 0.000} C_DIS
LIN {X 84.549,Y -40.664,Z -122.710,A -90.000,B 90.000,C 0.000} C_DIS
LIN {X 84.599,Y -40.669,Z -122.940,A -90.000,B 90.000,C 0.000} C_DIS
LIN {X 84.644,Y -40.680,Z -123.226,A -90.000,B 90.000,C 0.000} C_DIS
LIN {X 84.996,Y -40.632,Z -124.668,A -90.000,B 90.000,C 0.000} C_DIS
LIN {X 85.034,Y -40.629,Z -124.863,A -90.000,B 90.000,C 0.000} C_DIS
LIN {X 85.071,Y -40.640,Z -125.126,A -90.000,B 90.000,C 0.000} C_DIS
LIN {X 85.100,Y -40.640,Z -125.362,A -90.000,B 90.000,C 0.000} C_DIS
LIN {X 85.133,Y -40.637,Z -125.638,A -90.000,B 90.000,C 0.000} C_DIS
LIN {X 85.195,Y -40.619,Z -126.187,A -90.000,B 90.000,C 0.000} C_DIS
LIN {X 85.224,Y -40.612,Z -126.532,A -90.000,B 90.000,C 0.000} C_DIS
LIN {X 85.230,Y -40.611,Z -126.650,A -90.000,B 90.000,C 0.000} C_DIS
LIN {X 85.251,Y -40.611,Z -127.457,A -90.000,B 90.000,C 0.000} C_DIS
LIN {X 85.269,Y -40.586,Z -128.544,A -90.000,B 90.000,C 0.000} C_DIS
LIN {X 85.268,Y -40.584,Z -128.673,A -90.000,B 90.000,C 0.000} C_DIS
LIN {X 85.241,Y -40.584,Z -129.294,A -90.000,B 90.000,C 0.000} C_DIS
LIN {X 85.236,Y -40.584,Z -129.453,A -90.000,B 90.000,C 0.000} C_DIS
LIN {X 85.198,Y -40.563,Z -130.739,A -90.000,B 90.000,C 0.000} C_DIS
LIN {X 85.189,Y -40.562,Z -130.925,A -90.000,B 90.000,C 0.000} C_DIS
LIN {X 85.135,Y -40.563,Z -131.677,A -90.000,B 90.000,C 0.000} C_DIS
LIN {X 85.087,Y -40.544,Z -133.070,A -90.000,B 90.000,C 0.000} C_DIS
LIN {X 85.079,Y -40.542,Z -133.246,A -90.000,B 90.000,C 0.000} C_DIS
LIN {X 85.016,Y -40.543,Z -134.189,A -90.000,B 90.000,C 0.000} C_DIS
LIN {X 84.984,Y -40.543,Z -134.955,A -90.000,B 90.000,C 0.000} C_DIS
LIN {X 84.956,Y -40.523,Z -136.834,A -90.000,B 90.000,C 0.000} C_DIS
LIN {X 84.952,Y -40.523,Z -137.108,A -90.000,B 90.000,C 0.000} C_DIS
LIN {X 84.912,Y -40.523,Z -138.260,A -90.000,B 90.000,C 0.000} C_DIS
LIN {X 84.880,Y -40.503,Z -140.455,A -90.000,B 90.000,C 0.000} C_DIS
LIN {X 84.807,Y -40.494,Z -142.058,A -90.000,B 90.000,C 0.000} C_DIS
LIN {X 84.747,Y -40.465,Z -144.052,A -90.000,B 90.000,C 0.000} C_DIS
LIN {X 84.713,Y -40.462,Z -144.606,A -90.000,B 90.000,C 0.000} C_DIS
LIN {X 84.607,Y -40.451,Z -146.238,A -90.000,B 90.000,C 0.000} C_DIS
LIN {X 84.514,Y -40.422,Z -147.937,A -90.000,B 90.000,C 0.000} C_DIS
LIN {X 84.483,Y -40.421,Z -148.265,A -90.000,B 90.000,C 0.000} C_DIS
LIN {X 84.263,Y -40.397,Z -150.564,A -90.000,B 90.000,C 0.000} C_DIS
LIN {X 84.216,Y -40.389,Z -151.098,A -90.000,B 90.000,C 0.000} C_DIS
LIN {X 84.159,Y -40.378,Z -151.746,A -90.000,B 90.000,C 0.000} C_DIS
LIN {X 84.121,Y -40.374,Z -152.098,A -90.000,B 90.000,C 0.000} C_DIS
LIN {X 83.749,Y -40.347,Z -154.935,A -90.000,B 90.000,C 0.000} C_DIS
LIN {X 83.626,Y -40.331,Z -155.882,A -90.000,B 90.000,C 0.000} C_DIS
LIN {X 83.605,Y -40.328,Z -156.021,A -90.000,B 90.000,C 0.000} C_DIS
LIN {X 83.214,Y -40.311,Z -158.285,A -90.000,B 90.000,C 0.000} C_DIS
LIN {X 82.984,Y -40.296,Z -159.604,A -90.000,B 90.000,C 0.000} C_DIS
LIN {X 82.957,Y -40.291,Z -159.754,A -90.000,B 90.000,C 0.000} C_DIS
LIN {X 82.938,Y -40.290,Z -159.848,A -90.000,B 90.000,C 0.000} C_DIS
LIN {X 82.481,Y -40.283,Z -161.903,A -90.000,B 90.000,C 0.000} C_DIS
LIN {X 82.134,Y -40.272,Z -163.449,A -90.000,B 90.000,C 0.000} C_DIS
LIN {X 82.103,Y -40.272,Z -163.575,A -90.000,B 90.000,C 0.000} C_DIS
LIN {X 82.024,Y -40.270,Z -163.869,A -90.000,B 90.000,C 0.000} C_DIS
LIN {X 81.656,Y -40.274,Z -165.173,A -90.000,B 90.000,C 0.000} C_DIS
LIN {X 81.113,Y -40.278,Z -167.091,A -90.000,B 90.000,C 0.000} C_DIS
LIN {X 81.024,Y -40.275,Z -167.396,A -90.000,B 90.000,C 0.000} C_DIS
LIN {X 80.166,Y -40.292,Z -170.082,A -90.000,B 90.000,C 0.000} C_DIS
LIN {X 79.932,Y -40.295,Z -170.807,A -90.000,B 90.000,C 0.000} C_DIS
LIN {X 79.572,Y -40.303,Z -171.891,A -90.000,B 90.000,C 0.000} C_DIS
LIN {X 78.974,Y -40.315,Z -173.692,A -90.000,B 90.000,C 0.000} C_DIS
LIN {X 78.869,Y -40.318,Z -174.010,A -90.000,B 90.000,C 0.000} C_DIS
LIN {X 78.399,Y -40.323,Z -175.501,A -90.000,B 90.000,C 0.000} C_DIS
LIN {X 78.003,Y -40.325,Z -176.755,A -90.000,B 90.000,C 0.000} C_DIS
LIN {X 77.938,Y -40.328,Z -176.965,A -90.000,B 90.000,C 0.000} C_DIS
LIN {X 77.856,Y -40.324,Z -177.272,A -90.000,B 90.000,C 0.000} C_DIS
LIN {X 77.401,Y -40.314,Z -178.986,A -90.000,B 90.000,C 0.000} C_DIS
LIN {X 77.275,Y -40.310,Z -179.473,A -90.000,B 90.000,C 0.000} C_DIS
LIN {X 77.199,Y -40.303,Z -179.797,A -90.000,B 90.000,C 0.000} C_DIS
LIN {X 76.723,Y -40.276,Z -181.885,A -90.000,B 90.000,C 0.000} C_DIS
LIN {X 76.655,Y -40.270,Z -182.193,A -90.000,B 90.000,C 0.000} C_DIS
LIN {X 76.526,Y -40.253,Z -182.799,A -90.000,B 90.000,C 0.000} C_DIS
LIN {X 76.113,Y -40.216,Z -184.790,A -90.000,B 90.000,C 0.000} C_DIS
LIN {X 76.030,Y -40.204,Z -185.192,A -90.000,B 90.000,C 0.000} C_DIS
LIN {X 75.913,Y -40.190,Z -185.728,A -90.000,B 90.000,C 0.000} C_DIS
LIN {X 75.561,Y -40.166,Z -187.390,A -90.000,B 90.000,C 0.000} C_DIS
LIN {X 75.298,Y -40.137,Z -188.527,A -90.000,B 90.000,C 0.000} C_DIS
LIN {X 75.218,Y -40.132,Z -188.885,A -90.000,B 90.000,C 0.000} C_DIS
LIN {X 74.974,Y -40.127,Z -189.907,A -90.000,B 90.000,C 0.000} C_DIS
LIN {X 74.895,Y -40.121,Z -190.213,A -90.000,B 90.000,C 0.000} C_DIS
LIN {X 74.610,Y -40.106,Z -191.263,A -90.000,B 90.000,C 0.000} C_DIS
LIN {X 74.289,Y -40.101,Z -192.473,A -90.000,B 90.000,C 0.000} C_DIS
LIN {X 74.245,Y -40.099,Z -192.634,A -90.000,B 90.000,C 0.000} C_DIS
LIN {X 74.187,Y -40.098,Z -192.839,A -90.000,B 90.000,C 0.000} C_DIS
LIN {X 73.738,Y -40.082,Z -194.317,A -90.000,B 90.000,C 0.000} C_DIS
LIN {X 73.585,Y -40.078,Z -194.826,A -90.000,B 90.000,C 0.000} C_DIS
LIN {X 73.327,Y -40.078,Z -195.678,A -90.000,B 90.000,C 0.000} C_DIS
LIN {X 73.258,Y -40.073,Z -195.893,A -90.000,B 90.000,C 0.000} C_DIS
LIN {X 72.596,Y -40.064,Z -197.840,A -90.000,B 90.000,C 0.000} C_DIS
LIN {X 72.219,Y -40.064,Z -198.961,A -90.000,B 90.000,C 0.000} C_DIS
LIN {X 72.134,Y -40.060,Z -199.204,A -90.000,B 90.000,C 0.000} C_DIS
LIN {X 71.214,Y -40.053,Z -201.706,A -90.000,B 90.000,C 0.000} C_DIS
LIN {X 71.059,Y -40.053,Z -202.131,A -90.000,B 90.000,C 0.000} C_DIS
LIN {X 70.791,Y -40.053,Z -202.863,A -90.000,B 90.000,C 0.000} C_DIS
LIN {X 70.695,Y -40.050,Z -203.121,A -90.000,B 90.000,C 0.000} C_DIS
LIN {X 69.528,Y -40.046,Z -206.122,A -90.000,B 90.000,C 0.000} C_DIS
LIN {X 69.085,Y -40.046,Z -207.265,A -90.000,B 90.000,C 0.000} C_DIS
LIN {X 68.954,Y -40.044,Z -207.595,A -90.000,B 90.000,C 0.000} C_DIS
LIN {X 68.699,Y -40.043,Z -208.219,A -90.000,B 90.000,C 0.000} C_DIS
LIN {X 67.142,Y -40.040,Z -212.048,A -90.000,B 90.000,C 0.000} C_DIS
LIN {X 67.033,Y -40.038,Z -212.310,A -90.000,B 90.000,C 0.000} C_DIS
LIN {X 66.607,Y -40.038,Z -213.309,A -90.000,B 90.000,C 0.000} C_DIS
LIN {X 65.000,Y -40.035,Z -217.092,A -90.000,B 90.000,C 0.000} C_DIS
LIN {X 64.886,Y -40.033,Z -217.357,A -90.000,B 90.000,C 0.000} C_DIS
LIN {X 64.627,Y -40.033,Z -217.942,A -90.000,B 90.000,C 0.000} C_DIS
LIN {X 63.259,Y -40.028,Z -221.027,A -90.000,B 90.000,C 0.000} C_DIS
LIN {X 62.547,Y -40.028,Z -222.627,A -90.000,B 90.000,C 0.000} C_DIS
LIN {X 62.421,Y -40.024,Z -222.903,A -90.000,B 90.000,C 0.000} C_DIS
LIN {X 60.055,Y -40.026,Z -227.904,A -90.000,B 90.000,C 0.000} C_DIS
LIN {X 59.912,Y -40.020,Z -228.195,A -90.000,B 90.000,C 0.000} C_DIS
LIN {X 59.788,Y -40.020,Z -228.435,A -90.000,B 90.000,C 0.000} C_DIS
LIN {X 58.062,Y -40.038,Z -231.797,A -90.000,B 90.000,C 0.000} C_DIS
LIN {X 57.335,Y -40.038,Z -233.234,A -90.000,B 90.000,C 0.000} C_DIS
LIN {X 57.170,Y -40.029,Z -233.542,A -90.000,B 90.000,C 0.000} C_DIS
LIN {X 57.128,Y -40.027,Z -233.617,A -90.000,B 90.000,C 0.000} C_DIS
LIN {X 55.144,Y -40.070,Z -237.121,A -90.000,B 90.000,C 0.000} C_DIS
LIN {X 54.350,Y -40.070,Z -238.567,A -90.000,B 90.000,C 0.000} C_DIS
LIN {X 54.164,Y -40.063,Z -238.894,A -90.000,B 90.000,C 0.000} C_DIS
LIN {X 53.159,Y -40.062,Z -240.567,A -90.000,B 90.000,C 0.000} C_DIS
LIN {X 52.853,Y -40.064,Z -241.073,A -90.000,B 90.000,C 0.000} C_DIS
LIN {X 51.316,Y -40.122,Z -243.484,A -90.000,B 90.000,C 0.000} C_DIS
LIN {X 51.265,Y -40.122,Z -243.561,A -90.000,B 90.000,C 0.000} C_DIS
LIN {X 51.265,Y -60.000,Z -243.561,A -90.000,B 90.000,C 0.000} C_DIS
LIN {X -34.282,Y -60.000,Z -217.500,A -90.000,B 90.000,C 0.000} C_DIS
LIN {X -34.282,Y -39.308,Z -217.500,A -90.000,B 90.000,C 0.000} C_DIS
LIN {X -33.458,Y -39.327,Z -217.125,A -90.000,B 90.000,C 0.000} C_DIS
LIN {X -32.716,Y -39.350,Z -216.782,A -90.000,B 90.000,C 0.000} C_DIS
LIN {X -32.400,Y -39.362,Z -216.640,A -90.000,B 90.000,C 0.000} C_DIS
LIN {X -31.672,Y -39.382,Z -216.317,A -90.000,B 90.000,C 0.000} C_DIS
LIN {X -28.583,Y -39.418,Z -214.849,A -90.000,B 90.000,C 0.000} C_DIS
LIN {X -27.271,Y -39.434,Z -214.222,A -90.000,B 90.000,C 0.000} C_DIS
LIN {X -25.511,Y -39.476,Z -213.368,A -90.000,B 90.000,C 0.000} C_DIS
LIN {X -24.735,Y -39.487,Z -212.964,A -90.000,B 90.000,C 0.000} C_DIS
LIN {X -22.698,Y -39.503,Z -211.879,A -90.000,B 90.000,C 0.000} C_DIS
LIN {X -22.257,Y -39.515,Z -211.660,A -90.000,B 90.000,C 0.000} C_DIS
LIN {X -21.775,Y -39.533,Z -211.417,A -90.000,B 90.000,C 0.000} C_DIS
LIN {X -20.722,Y -39.583,Z -210.882,A -90.000,B 90.000,C 0.000} C_DIS
LIN {X -20.445,Y -39.595,Z -210.746,A -90.000,B 90.000,C 0.000} C_DIS
LIN {X -18.691,Y -39.633,Z -209.790,A -90.000,B 90.000,C 0.000} C_DIS
LIN {X -17.711,Y -39.646,Z -209.261,A -90.000,B 90.000,C 0.000} C_DIS
LIN {X -17.437,Y -39.655,Z -209.110,A -90.000,B 90.000,C 0.000} C_DIS
LIN {X -15.943,Y -39.691,Z -208.252,A -90.000,B 90.000,C 0.000} C_DIS
LIN {X -14.848,Y -39.703,Z -207.588,A -90.000,B 90.000,C 0.000} C_DIS
LIN {X -14.383,Y -39.711,Z -207.304,A -90.000,B 90.000,C 0.000} C_DIS
LIN {X -13.461,Y -39.718,Z -206.719,A -90.000,B 90.000,C 0.000} C_DIS
LIN {X -13.222,Y -39.723,Z -206.565,A -90.000,B 90.000,C 0.000} C_DIS
LIN {X -11.806,Y -39.753,Z -205.655,A -90.000,B 90.000,C 0.000} C_DIS
LIN {X -9.716,Y -39.769,Z -204.243,A -90.000,B 90.000,C 0.000} C_DIS
LIN {X -9.607,Y -39.771,Z -204.173,A -90.000,B 90.000,C 0.000} C_DIS
LIN {X -9.379,Y -39.778,Z -204.032,A -90.000,B 90.000,C 0.000} C_DIS
LIN {X -7.645,Y -39.858,Z -202.942,A -90.000,B 90.000,C 0.000} C_DIS
LIN {X -6.436,Y -39.873,Z -202.073,A -90.000,B 90.000,C 0.000} C_DIS
LIN {X -5.907,Y -39.880,Z -201.708,A -90.000,B 90.000,C 0.000} C_DIS
LIN {X -5.399,Y -39.886,Z -201.358,A -90.000,B 90.000,C 0.000} C_DIS
LIN {X -3.925,Y -39.931,Z -200.330,A -90.000,B 90.000,C 0.000} C_DIS
LIN {X -1.840,Y -39.911,Z -198.626,A -90.000,B 90.000,C 0.000} C_DIS
LIN {X -1.323,Y -39.922,Z -198.196,A -90.000,B 90.000,C 0.000} C_DIS
LIN {X -0.473,Y -39.942,Z -197.524,A -90.000,B 90.000,C 0.000} C_DIS
LIN {X 1.807,Y -39.887,Z -195.383,A -90.000,B 90.000,C 0.000} C_DIS
LIN {X 2.700,Y -39.883,Z -194.536,A -90.000,B 90.000,C 0.000} C_DIS
LIN {X 2.903,Y -39.885,Z -194.352,A -90.000,B 90.000,C 0.000} C_DIS
LIN {X 3.793,Y -39.848,Z -193.396,A -90.000,B 90.000,C 0.000} C_DIS
LIN {X 5.311,Y -39.811,Z -191.747,A -90.000,B 90.000,C 0.000} C_DIS
LIN {X 5.929,Y -39.793,Z -191.081,A -90.000,B 90.000,C 0.000} C_DIS
LIN {X 7.176,Y -39.731,Z -189.661,A -90.000,B 90.000,C 0.000} C_DIS
LIN {X 8.435,Y -39.695,Z -188.208,A -90.000,B 90.000,C 0.000} C_DIS
LIN {X 8.784,Y -39.678,Z -187.811,A -90.000,B 90.000,C 0.000} C_DIS
LIN {X 10.549,Y -39.588,Z -185.776,A -90.000,B 90.000,C 0.000} C_DIS
LIN {X 11.343,Y -39.565,Z -184.849,A -90.000,B 90.000,C 0.000} C_DIS
LIN {X 11.738,Y -39.543,Z -184.397,A -90.000,B 90.000,C 0.000} C_DIS
LIN {X 11.891,Y -39.533,Z -184.219,A -90.000,B 90.000,C 0.000} C_DIS
LIN {X 13.120,Y -39.480,Z -182.855,A -90.000,B 90.000,C 0.000} C_DIS
LIN {X 13.268,Y -39.474,Z -182.691,A -90.000,B 90.000,C 0.000} C_DIS
LIN {X 14.112,Y -39.453,Z -181.742,A -90.000,B 90.000,C 0.000} C_DIS
LIN {X 14.527,Y -39.433,Z -181.283,A -90.000,B 90.000,C 0.000} C_DIS
LIN {X 14.646,Y -39.425,Z -181.148,A -90.000,B 90.000,C 0.000} C_DIS
LIN {X 14.874,Y -39.413,Z -180.895,A -90.000,B 90.000,C 0.000} C_DIS
LIN {X 15.026,Y -39.408,Z -180.733,A -90.000,B 90.000,C 0.000} C_DIS
LIN {X 15.366,Y -39.401,Z -180.389,A -90.000,B 90.000,C 0.000} C_DIS
LIN {X 17.020,Y -39.360,Z -178.718,A -90.000,B 90.000,C 0.000} C_DIS
LIN {X 17.573,Y -39.344,Z -178.163,A -90.000,B 90.000,C 0.000} C_DIS
LIN {X 17.794,Y -39.339,Z -177.946,A -90.000,B 90.000,C 0.000} C_DIS
LIN {X 19.881,Y -39.319,Z -175.954,A -90.000,B 90.000,C 0.000} C_DIS
LIN {X 20.993,Y -39.308,Z -174.878,A -90.000,B 90.000,C 0.000} C_DIS
LIN {X 21.175,Y -39.312,Z -174.702,A -90.000,B 90.000,C 0.000} C_DIS
LIN {X 21.409,Y -39.308,Z -174.476,A -90.000,B 90.000,C 0.000} C_DIS
LIN {X 21.924,Y -39.315,Z -173.983,A -90.000,B 90.000,C 0.000} C_DIS
LIN {X 22.750,Y -39.313,Z -173.143,A -90.000,B 90.000,C 0.000} C_DIS
LIN {X 23.522,Y -39.330,Z -172.344,A -90.000,B 90.000,C 0.000} C_DIS
LIN {X 23.756,Y -39.328,Z -172.079,A -90.000,B 90.000,C 0.000} C_DIS
LIN {X 24.424,Y -39.322,Z -171.309,A -90.000,B 90.000,C 0.000} C_DIS
LIN {X 24.973,Y -39.332,Z -170.664,A -90.000,B 90.000,C 0.000} C_DIS
LIN {X 25.295,Y -39.326,Z -170.245,A -90.000,B 90.000,C 0.000} C_DIS
LIN {X 25.862,Y -39.321,Z -169.520,A -90.000,B 90.000,C 0.000} C_DIS
LIN {X 26.233,Y -39.324,Z -169.039,A -90.000,B 90.000,C 0.000} C_DIS
LIN {X 26.804,Y -39.308,Z -168.223,A -90.000,B 90.000,C 0.000} C_DIS
LIN {X 26.804,Y -60.000,Z -168.223,A -90.000,B 90.000,C 0.000} C_DIS
LIN {X 34.198,Y -60.000,Z -155.287,A -90.000,B 90.000,C 0.000} C_DIS
LIN {X 34.198,Y -39.308,Z -155.287,A -90.000,B 90.000,C 0.000} C_DIS
LIN {X 34.301,Y -39.335,Z -155.023,A -90.000,B 90.000,C 0.000} C_DIS
LIN {X 34.402,Y -39.353,Z -154.768,A -90.000,B 90.000,C 0.000} C_DIS
LIN {X 34.636,Y -39.391,Z -154.184,A -90.000,B 90.000,C 0.000} C_DIS
LIN {X 34.811,Y -39.419,Z -153.770,A -90.000,B 90.000,C 0.000} C_DIS
LIN {X 34.967,Y -39.462,Z -153.386,A -90.000,B 90.000,C 0.000} C_DIS
LIN {X 35.057,Y -39.485,Z -153.168,A -90.000,B 90.000,C 0.000} C_DIS
LIN {X 35.122,Y -39.495,Z -153.016,A -90.000,B 90.000,C 0.000} C_DIS
LIN {X 35.189,Y -39.519,Z -152.825,A -90.000,B 90.000,C 0.000} C_DIS
LIN {X 35.401,Y -39.597,Z -152.208,A -90.000,B 90.000,C 0.000} C_DIS
LIN {X 35.472,Y -39.621,Z -152.011,A -90.000,B 90.000,C 0.000} C_DIS
LIN {X 35.540,Y -39.635,Z -151.829,A -90.000,B 90.000,C 0.000} C_DIS
LIN {X 35.586,Y -39.642,Z -151.708,A -90.000,B 90.000,C 0.000} C_DIS
LIN {X 35.878,Y -39.685,Z -151.002,A -90.000,B 90.000,C 0.000} C_DIS
LIN {X 36.028,Y -39.732,Z -150.630,A -90.000,B 90.000,C 0.000} C_DIS
LIN {X 36.097,Y -39.747,Z -150.465,A -90.000,B 90.000,C 0.000} C_DIS
LIN {X 36.175,Y -39.762,Z -150.245,A -90.000,B 90.000,C 0.000} C_DIS
LIN {X 36.334,Y -39.782,Z -149.802,A -90.000,B 90.000,C 0.000} C_DIS
LIN {X 36.398,Y -39.790,Z -149.641,A -90.000,B 90.000,C 0.000} C_DIS
LIN {X 36.471,Y -39.800,Z -149.468,A -90.000,B 90.000,C 0.000} C_DIS
LIN {X 36.646,Y -39.840,Z -149.045,A -90.000,B 90.000,C 0.000} C_DIS
LIN {X 36.919,Y -39.900,Z -148.406,A -90.000,B 90.000,C 0.000} C_DIS
LIN {X 36.982,Y -39.911,Z -148.262,A -90.000,B 90.000,C 0.000} C_DIS
LIN {X 37.058,Y -39.917,Z -148.091,A -90.000,B 90.000,C 0.000} C_DIS
LIN {X 37.166,Y -39.919,Z -147.847,A -90.000,B 90.000,C 0.000} C_DIS
LIN {X 37.268,Y -39.922,Z -147.610,A -90.000,B 90.000,C 0.000} C_DIS
LIN {X 37.296,Y -39.922,Z -147.550,A -90.000,B 90.000,C 0.000} C_DIS
LIN {X 37.366,Y -39.923,Z -147.380,A -90.000,B 90.000,C 0.000} C_DIS
LIN {X 37.468,Y -39.927,Z -147.159,A -90.000,B 90.000,C 0.000} C_DIS
LIN {X 37.728,Y -39.965,Z -146.604,A -90.000,B 90.000,C 0.000} C_DIS
LIN {X 37.838,Y -39.975,Z -146.363,A -90.000,B 90.000,C 0.000} C_DIS
LIN {X 37.943,Y -39.979,Z -146.134,A -90.000,B 90.000,C 0.000} C_DIS
LIN {X 38.200,Y -39.974,Z -145.585,A -90.000,B 90.000,C 0.000} C_DIS
LIN {X 38.385,Y -39.973,Z -145.203,A -90.000,B 90.000,C 0.000} C_DIS
LIN {X 38.575,Y -39.987,Z -144.849,A -90.000,B 90.000,C 0.000} C_DIS
LIN {X 38.816,Y -40.006,Z -144.414,A -90.000,B 90.000,C 0.000} C_DIS
LIN {X 38.888,Y -40.011,Z -144.270,A -90.000,B 90.000,C 0.000} C_DIS
LIN {X 39.142,Y -40.005,Z -143.766,A -90.000,B 90.000,C 0.000} C_DIS
LIN {X 39.433,Y -39.982,Z -143.201,A -90.000,B 90.000,C 0.000} C_DIS
LIN {X 39.524,Y -39.977,Z -143.040,A -90.000,B 90.000,C 0.000} C_DIS
LIN {X 39.625,Y -39.974,Z -142.875,A -90.000,B 90.000,C 0.000} C_DIS
LIN {X 39.739,Y -39.977,Z -142.693,A -90.000,B 90.000,C 0.000} C_DIS
LIN {X 40.096,Y -39.984,Z -142.140,A -90.000,B 90.000,C 0.000} C_DIS
LIN {X 40.630,Y -39.952,Z -141.336,A -90.000,B 90.000,C 0.000} C_DIS
LIN {X 40.730,Y -39.952,Z -141.182,A -90.000,B 90.000,C 0.000} C_DIS
LIN {X 41.064,Y -39.948,Z -140.644,A -90.000,B 90.000,C 0.000} C_DIS
LIN {X 41.213,Y -39.949,Z -140.424,A -90.000,B 90.000,C 0.000} C_DIS
LIN {X 41.511,Y -39.954,Z -140.013,A -90.000,B 90.000,C 0.000} C_DIS
LIN {X 41.683,Y -39.954,Z -139.761,A -90.000,B 90.000,C 0.000} C_DIS
LIN {X 41.794,Y -39.949,Z -139.600,A -90.000,B 90.000,C 0.000} C_DIS
LIN {X 42.531,Y -39.898,Z -138.547,A -90.000,B 90.000,C 0.000} C_DIS
LIN {X 42.595,Y -39.895,Z -138.460,A -90.000,B 90.000,C 0.000} C_DIS
LIN {X 42.661,Y -39.892,Z -138.375,A -90.000,B 90.000,C 0.000} C_DIS
LIN {X 43.012,Y -39.881,Z -137.950,A -90.000,B 90.000,C 0.000} C_DIS
LIN {X 43.417,Y -39.886,Z -137.448,A -90.000,B 90.000,C 0.000} C_DIS
LIN {X 43.584,Y -39.887,Z -137.243,A -90.000,B 90.000,C 0.000} C_DIS
LIN {X 43.848,Y -39.878,Z -136.921,A -90.000,B 90.000,C 0.000} C_DIS
LIN {X 44.344,Y -39.859,Z -136.304,A -90.000,B 90.000,C 0.000} C_DIS
LIN {X 44.408,Y -39.857,Z -136.228,A -90.000,B 90.000,C 0.000} C_DIS
LIN {X 44.783,Y -39.852,Z -135.803,A -90.000,B 90.000,C 0.000} C_DIS
LIN {X 45.171,Y -39.851,Z -135.363,A -90.000,B 90.000,C 0.000} C_DIS
LIN {X 45.982,Y -39.841,Z -134.399,A -90.000,B 90.000,C 0.000} C_DIS
LIN {X 46.347,Y -39.839,Z -133.976,A -90.000,B 90.000,C 0.000} C_DIS
LIN {X 46.988,Y -39.844,Z -133.266,A -90.000,B 90.000,C 0.000} C_DIS
LIN {X 47.291,Y -39.848,Z -132.931,A -90.000,B 90.000,C 0.000} C_DIS
LIN {X 48.271,Y -39.862,Z -131.854,A -90.000,B 90.000,C 0.000} C_DIS
LIN {X 48.489,Y -39.868,Z -131.626,A -90.000,B 90.000,C 0.000} C_DIS
LIN {X 48.959,Y -39.890,Z -131.126,A -90.000,B 90.000,C 0.000} C_DIS
LIN {X 51.568,Y -39.950,Z -128.042,A -90.000,B 90.000,C 0.000} C_DIS
LIN {X 51.632,Y -39.953,Z -127.966,A -90.000,B 90.000,C 0.000} C_DIS
LIN {X 51.706,Y -39.958,Z -127.877,A -90.000,B 90.000,C 0.000} C_DIS
LIN {X 53.142,Y -39.959,Z -125.591,A -90.000,B 90.000,C 0.000} C_DIS
LIN {X 53.556,Y -39.956,Z -124.915,A -90.000,B 90.000,C 0.000} C_DIS
LIN {X 54.095,Y -39.943,Z -123.980,A -90.000,B 90.000,C 0.000} C_DIS
LIN {X 54.466,Y -39.934,Z -123.337,A -90.000,B 90.000,C 0.000} C_DIS
LIN {X 55.483,Y -39.882,Z -121.445,A -90.000,B 90.000,C 0.000} C_DIS
LIN {X 55.703,Y -39.871,Z -121.034,A -90.000,B 90.000,C 0.000} C_DIS
LIN {X 55.774,Y -39.870,Z -120.913,A -90.000,B 90.000,C 0.000} C_DIS
LIN {X 55.823,Y -39.869,Z -120.833,A -90.000,B 90.000,C 0.000} C_DIS
LIN {X 55.841,Y -39.868,Z -120.794,A -90.000,B 90.000,C 0.000} C_DIS
LIN {X 56.243,Y -39.854,Z -120.086,A -90.000,B 90.000,C 0.000} C_DIS
LIN {X 56.441,Y -39.846,Z -119.740,A -90.000,B 90.000,C 0.000} C_DIS
LIN {X 57.375,Y -39.824,Z -118.095,A -90.000,B 90.000,C 0.000} C_DIS
LIN {X 58.038,Y -39.804,Z -116.932,A -90.000,B 90.000,C 0.000} C_DIS
LIN {X 58.369,Y -39.783,Z -116.304,A -90.000,B 90.000,C 0.000} C_DIS
LIN {X 58.541,Y -39.776,Z -115.974,A -90.000,B 90.000,C 0.000} C_DIS
LIN {X 59.408,Y -39.748,Z -114.370,A -90.000,B 90.000,C 0.000} C_DIS
LIN {X 59.824,Y -39.743,Z -113.591,A -90.000,B 90.000,C 0.000} C_DIS
LIN {X 60.135,Y -39.733,Z -113.015,A -90.000,B 90.000,C 0.000} C_DIS
LIN {X 60.309,Y -39.726,Z -112.686,A -90.000,B 90.000,C 0.000} C_DIS
LIN {X 60.465,Y -39.730,Z -112.380,A -90.000,B 90.000,C 0.000} C_DIS
LIN {X 60.634,Y -39.735,Z -112.050,A -90.000,B 90.000,C 0.000} C_DIS
LIN {X 61.631,Y -39.724,Z -109.871,A -90.000,B 90.000,C 0.000} C_DIS
LIN {X 61.684,Y -39.722,Z -109.750,A -90.000,B 90.000,C 0.000} C_DIS
LIN {X 61.848,Y -39.722,Z -109.403,A -90.000,B 90.000,C 0.000} C_DIS
LIN {X 62.816,Y -39.804,Z -107.291,A -90.000,B 90.000,C 0.000} C_DIS
LIN {X 62.997,Y -39.823,Z -106.900,A -90.000,B 90.000,C 0.000} C_DIS
LIN {X 63.215,Y -39.844,Z -106.376,A -90.000,B 90.000,C 0.000} C_DIS
LIN {X 63.451,Y -39.896,Z -105.781,A -90.000,B 90.000,C 0.000} C_DIS
LIN {X 63.616,Y -39.930,Z -105.291,A -90.000,B 90.000,C 0.000} C_DIS
LIN {X 64.000,Y -39.999,Z -104.162,A -90.000,B 90.000,C 0.000} C_DIS
LIN {X 64.135,Y -40.019,Z -103.596,A -90.000,B 90.000,C 0.000} C_DIS
LIN {X 64.174,Y -40.035,Z -103.421,A -90.000,B 90.000,C 0.000} C_DIS
LIN {X 64.338,Y -40.099,Z -102.775,A -90.000,B 90.000,C 0.000} C_DIS
LIN {X 64.418,Y -40.138,Z -102.146,A -90.000,B 90.000,C 0.000} C_DIS
LIN {X 64.409,Y -40.142,Z -101.901,A -90.000,B 90.000,C 0.000} C_DIS
LIN {X 64.367,Y -40.134,Z -101.767,A -90.000,B 90.000,C 0.000} C_DIS
LIN {X 64.035,Y -40.125,Z -100.766,A -90.000,B 90.000,C 0.000} C_DIS
LIN {X 63.977,Y -40.119,Z -100.654,A -90.000,B 90.000,C 0.000} C_DIS
LIN {X 63.550,Y -40.103,Z -99.840,A -90.000,B 90.000,C 0.000} C_DIS
LIN {X 63.216,Y -40.098,Z -99.211,A -90.000,B 90.000,C 0.000} C_DIS
LIN {X 63.010,Y -40.105,Z -98.826,A -90.000,B 90.000,C 0.000} C_DIS
LIN {X 62.826,Y -40.114,Z -98.455,A -90.000,B 90.000,C 0.000} C_DIS
LIN {X 62.450,Y -40.177,Z -97.721,A -90.000,B 90.000,C 0.000} C_DIS
LIN {X 62.408,Y -40.183,Z -97.637,A -90.000,B 90.000,C 0.000} C_DIS
LIN {X 62.339,Y -40.187,Z -97.497,A -90.000,B 90.000,C 0.000} C_DIS
LIN {X 62.222,Y -40.183,Z -97.249,A -90.000,B 90.000,C 0.000} C_DIS
LIN {X 62.004,Y -40.174,Z -96.745,A -90.000,B 90.000,C 0.000} C_DIS
LIN {X 61.945,Y -40.188,Z -96.617,A -90.000,B 90.000,C 0.000} C_DIS
LIN {X 61.890,Y -40.199,Z -96.497,A -90.000,B 90.000,C 0.000} C_DIS
LIN {X 61.779,Y -40.222,Z -96.221,A -90.000,B 90.000,C 0.000} C_DIS
LIN {X 61.727,Y -40.226,Z -96.068,A -90.000,B 90.000,C 0.000} C_DIS
LIN {X 61.658,Y -40.224,Z -95.854,A -90.000,B 90.000,C 0.000} C_DIS
LIN {X 61.599,Y -40.222,Z -95.645,A -90.000,B 90.000,C 0.000} C_DIS
LIN {X 61.424,Y -40.217,Z -94.943,A -90.000,B 90.000,C 0.000} C_DIS
LIN {X 61.280,Y -40.243,Z -94.391,A -90.000,B 90.000,C 0.000} C_DIS
LIN {X 61.231,Y -40.245,Z -94.195,A -90.000,B 90.000,C 0.000} C_DIS
LIN {X 61.187,Y -40.238,Z -94.015,A -90.000,B 90.000,C 0.000} C_DIS
LIN {X 61.154,Y -40.229,Z -93.878,A -90.000,B 90.000,C 0.000} C_DIS
LIN {X 60.911,Y -40.259,Z -92.932,A -90.000,B 90.000,C 0.000} C_DIS
LIN {X 60.893,Y -40.262,Z -92.849,A -90.000,B 90.000,C 0.000} C_DIS
LIN {X 60.851,Y -40.265,Z -92.626,A -90.000,B 90.000,C 0.000} C_DIS
LIN {X 60.838,Y -40.263,Z -92.544,A -90.000,B 90.000,C 0.000} C_DIS
LIN {X 60.776,Y -40.230,Z -92.008,A -90.000,B 90.000,C 0.000} C_DIS
LIN {X 60.762,Y -40.220,Z -91.847,A -90.000,B 90.000,C 0.000} C_DIS
LIN {X 60.755,Y -40.204,Z -91.569,A -90.000,B 90.000,C 0.000} C_DIS
LIN {X 60.759,Y -40.176,Z -91.047,A -90.000,B 90.000,C 0.000} C_DIS
LIN {X 60.754,Y -40.173,Z -90.561,A -90.000,B 90.000,C 0.000} C_DIS
LIN {X 60.755,Y -40.160,Z -90.346,A -90.000,B 90.000,C 0.000} C_DIS
LIN {X 60.753,Y -40.160,Z -90.167,A -90.000,B 90.000,C 0.000} C_DIS
LIN {X 60.752,Y -40.156,Z -90.036,A -90.000,B 90.000,C 0.000} C_DIS
LIN {X 60.753,Y -40.136,Z -89.695,A -90.000,B 90.000,C 0.000} C_DIS
LIN {X 60.750,Y -40.125,Z -88.217,A -90.000,B 90.000,C 0.000} C_DIS
LIN {X 60.754,Y -40.109,Z -87.968,A -90.000,B 90.000,C 0.000} C_DIS
LIN {X 60.775,Y -40.082,Z -87.522,A -90.000,B 90.000,C 0.000} C_DIS
LIN {X 60.805,Y -40.050,Z -87.011,A -90.000,B 90.000,C 0.000} C_DIS
LIN {X 60.843,Y -40.069,Z -86.017,A -90.000,B 90.000,C 0.000} C_DIS
LIN {X 60.840,Y -40.070,Z -85.856,A -90.000,B 90.000,C 0.000} C_DIS
LIN {X 60.824,Y -40.031,Z -84.554,A -90.000,B 90.000,C 0.000} C_DIS
LIN {X 60.825,Y -40.028,Z -84.447,A -90.000,B 90.000,C 0.000} C_DIS
LIN {X 60.831,Y -40.025,Z -84.304,A -90.000,B 90.000,C 0.000} C_DIS
LIN {X 60.836,Y -40.029,Z -84.149,A -90.000,B 90.000,C 0.000} C_DIS
LIN {X 60.841,Y -40.041,Z -83.999,A -90.000,B 90.000,C 0.000} C_DIS
LIN {X 60.853,Y -40.055,Z -83.801,A -90.000,B 90.000,C 0.000} C_DIS
LIN {X 60.846,Y -40.080,Z -83.306,A -90.000,B 90.000,C 0.000} C_DIS
LIN {X 60.824,Y -40.155,Z -82.613,A -90.000,B 90.000,C 0.000} C_DIS
LIN {X 60.727,Y -40.266,Z -81.529,A -90.000,B 90.000,C 0.000} C_DIS
LIN {X 60.712,Y -40.289,Z -81.373,A -90.000,B 90.000,C 0.000} C_DIS
LIN {X 60.609,Y -40.326,Z -81.028,A -90.000,B 90.000,C 0.000} C_DIS
LIN {X 60.570,Y -40.343,Z -80.882,A -90.000,B 90.000,C 0.000} C_DIS
LIN {X 60.537,Y -40.360,Z -80.743,A -90.000,B 90.000,C 0.000} C_DIS
LIN {X 60.503,Y -40.382,Z -80.567,A -90.000,B 90.000,C 0.000} C_DIS
LIN {X 60.441,Y -40.435,Z -80.173,A -90.000,B 90.000,C 0.000} C_DIS
LIN {X 60.427,Y -40.451,Z -80.052,A -90.000,B 90.000,C 0.000} C_DIS
LIN {X 60.348,Y -40.578,Z -79.414,A -90.000,B 90.000,C 0.000} C_DIS
LIN {X 59.512,Y -40.485,Z -79.496,A -90.000,B 90.000,C 0.000} C_DIS
LIN {X 59.301,Y -40.470,Z -79.511,A -90.000,B 90.000,C 0.000} C_DIS
LIN {X 59.123,Y -40.458,Z -79.516,A -90.000,B 90.000,C 0.000} C_DIS
LIN {X 58.566,Y -40.424,Z -79.516,A -90.000,B 90.000,C 0.000} C_DIS
LIN {X 58.357,Y -40.403,Z -79.557,A -90.000,B 90.000,C 0.000} C_DIS
LIN {X 58.149,Y -40.392,Z -79.600,A -90.000,B 90.000,C 0.000} C_DIS
LIN {X 57.290,Y -40.401,Z -79.790,A -90.000,B 90.000,C 0.000} C_DIS
LIN {X 56.589,Y -40.411,Z -79.929,A -90.000,B 90.000,C 0.000} C_DIS
LIN {X 56.379,Y -40.419,Z -79.972,A -90.000,B 90.000,C 0.000} C_DIS
LIN {X 55.615,Y -40.430,Z -80.247,A -90.000,B 90.000,C 0.000} C_DIS
LIN {X 55.324,Y -40.435,Z -80.347,A -90.000,B 90.000,C 0.000} C_DIS
LIN {X 54.879,Y -40.443,Z -80.498,A -90.000,B 90.000,C 0.000} C_DIS
LIN {X 53.899,Y -40.568,Z -80.847,A -90.000,B 90.000,C 0.000} C_DIS
LIN {X 52.822,Y -40.698,Z -81.223,A -90.000,B 90.000,C 0.000} C_DIS
LIN {X 52.174,Y -40.776,Z -81.434,A -90.000,B 90.000,C 0.000} C_DIS
LIN {X 52.122,Y -40.782,Z -81.455,A -90.000,B 90.000,C 0.000} C_DIS
LIN {X 52.136,Y -40.782,Z -81.533,A -90.000,B 90.000,C 0.000} C_DIS
LIN {X 52.192,Y -40.776,Z -81.625,A -90.000,B 90.000,C 0.000} C_DIS
LIN {X 52.294,Y -40.767,Z -81.801,A -90.000,B 90.000,C 0.000} C_DIS
LIN {X 52.340,Y -40.760,Z -81.886,A -90.000,B 90.000,C 0.000} C_DIS
LIN {X 52.771,Y -40.681,Z -82.737,A -90.000,B 90.000,C 0.000} C_DIS
LIN {X 53.044,Y -40.680,Z -83.261,A -90.000,B 90.000,C 0.000} C_DIS
LIN {X 53.153,Y -40.673,Z -83.412,A -90.000,B 90.000,C 0.000} C_DIS
LIN {X 53.577,Y -40.641,Z -84.004,A -90.000,B 90.000,C 0.000} C_DIS
LIN {X 54.053,Y -40.615,Z -84.666,A -90.000,B 90.000,C 0.000} C_DIS
LIN {X 54.120,Y -40.611,Z -84.766,A -90.000,B 90.000,C 0.000} C_DIS
LIN {X 54.201,Y -40.608,Z -84.895,A -90.000,B 90.000,C 0.000} C_DIS
LIN {X 54.292,Y -40.604,Z -85.052,A -90.000,B 90.000,C 0.000} C_DIS
LIN {X 54.925,Y -40.556,Z -86.165,A -90.000,B 90.000,C 0.000} C_DIS
LIN {X 54.958,Y -40.553,Z -86.206,A -90.000,B 90.000,C 0.000} C_DIS
LIN {X 55.032,Y -40.550,Z -86.302,A -90.000,B 90.000,C 0.000} C_DIS
LIN {X 55.171,Y -40.546,Z -86.494,A -90.000,B 90.000,C 0.000} C_DIS
LIN {X 55.263,Y -40.545,Z -86.631,A -90.000,B 90.000,C 0.000} C_DIS
LIN {X 55.417,Y -40.540,Z -86.873,A -90.000,B 90.000,C 0.000} C_DIS
LIN {X 55.621,Y -40.530,Z -87.196,A -90.000,B 90.000,C 0.000} C_DIS
LIN {X 56.441,Y -40.516,Z -88.484,A -90.000,B 90.000,C 0.000} C_DIS
LIN {X 56.609,Y -40.507,Z -88.773,A -90.000,B 90.000,C 0.000} C_DIS
LIN {X 56.712,Y -40.501,Z -88.964,A -90.000,B 90.000,C 0.000} C_DIS
LIN {X 56.772,Y -40.499,Z -89.087,A -90.000,B 90.000,C 0.000} C_DIS
LIN {X 57.228,Y -40.482,Z -90.093,A -90.000,B 90.000,C 0.000} C_DIS
LIN {X 57.365,Y -40.489,Z -90.389,A -90.000,B 90.000,C 0.000} C_DIS
LIN {X 57.439,Y -40.489,Z -90.550,A -90.000,B 90.000,C 0.000} C_DIS
LIN {X 57.644,Y -40.477,Z -91.006,A -90.000,B 90.000,C 0.000} C_DIS
LIN {X 57.699,Y -40.474,Z -91.117,A -90.000,B 90.000,C 0.000} C_DIS
LIN {X 57.742,Y -40.474,Z -91.216,A -90.000,B 90.000,C 0.000} C_DIS
LIN {X 57.845,Y -40.477,Z -91.469,A -90.000,B 90.000,C 0.000} C_DIS
LIN {X 57.894,Y -40.480,Z -91.605,A -90.000,B 90.000,C 0.000} C_DIS
LIN {X 58.007,Y -40.488,Z -91.952,A -90.000,B 90.000,C 0.000} C_DIS
LIN {X 58.191,Y -40.505,Z -92.562,A -90.000,B 90.000,C 0.000} C_DIS
LIN {X 58.262,Y -40.506,Z -92.805,A -90.000,B 90.000,C 0.000} C_DIS
LIN {X 58.547,Y -40.479,Z -93.790,A -90.000,B 90.000,C 0.000} C_DIS
LIN {X 58.781,Y -40.496,Z -94.578,A -90.000,B 90.000,C 0.000} C_DIS
LIN {X 58.826,Y -40.493,Z -94.733,A -90.000,B 90.000,C 0.000} C_DIS
LIN {X 59.141,Y -40.422,Z -95.860,A -90.000,B 90.000,C 0.000} C_DIS
LIN {X 59.287,Y -40.406,Z -96.374,A -90.000,B 90.000,C 0.000} C_DIS
LIN {X 59.317,Y -40.403,Z -96.500,A -90.000,B 90.000,C 0.000} C_DIS
LIN {X 59.366,Y -40.399,Z -96.746,A -90.000,B 90.000,C 0.000} C_DIS
LIN {X 59.400,Y -40.397,Z -96.988,A -90.000,B 90.000,C 0.000} C_DIS
LIN {X 59.417,Y -40.390,Z -97.132,A -90.000,B 90.000,C 0.000} C_DIS
LIN {X 59.442,Y -40.370,Z -97.422,A -90.000,B 90.000,C 0.000} C_DIS
LIN {X 59.450,Y -40.360,Z -97.586,A -90.000,B 90.000,C 0.000} C_DIS
LIN {X 59.488,Y -40.326,Z -98.091,A -90.000,B 90.000,C 0.000} C_DIS
LIN {X 59.524,Y -40.316,Z -98.528,A -90.000,B 90.000,C 0.000} C_DIS
LIN {X 59.533,Y -40.311,Z -98.748,A -90.000,B 90.000,C 0.000} C_DIS
LIN {X 59.552,Y -40.272,Z -99.440,A -90.000,B 90.000,C 0.000} C_DIS
LIN {X 59.561,Y -40.227,Z -99.905,A -90.000,B 90.000,C 0.000} C_DIS
LIN {X 59.602,Y -40.149,Z -101.391,A -90.000,B 90.000,C 0.000} C_DIS
LIN {X 59.600,Y -40.137,Z -101.557,A -90.000,B 90.000,C 0.000} C_DIS
LIN {X 59.586,Y -40.119,Z -101.825,A -90.000,B 90.000,C 0.000} C_DIS
LIN {X 59.569,Y -40.107,Z -102.028,A -90.000,B 90.000,C 0.000} C_DIS
LIN {X 59.560,Y -40.103,Z -102.108,A -90.000,B 90.000,C 0.000} C_DIS
LIN {X 59.397,Y -40.005,Z -103.434,A -90.000,B 90.000,C 0.000} C_DIS
LIN {X 59.276,Y -39.964,Z -104.527,A -90.000,B 90.000,C 0.000} C_DIS
LIN {X 59.189,Y -39.854,Z -105.644,A -90.000,B 90.000,C 0.000} C_DIS
LIN {X 59.153,Y -39.832,Z -105.916,A -90.000,B 90.000,C 0.000} C_DIS
LIN {X 59.136,Y -39.824,Z -106.027,A -90.000,B 90.000,C 0.000} C_DIS
LIN {X 58.925,Y -39.765,Z -107.167,A -90.000,B 90.000,C 0.000} C_DIS
LIN {X 58.909,Y -39.759,Z -107.251,A -90.000,B 90.000,C 0.000} C_DIS
LIN {X 58.856,Y -39.747,Z -107.542,A -90.000,B 90.000,C 0.000} C_DIS
LIN {X 58.805,Y -39.736,Z -107.817,A -90.000,B 90.000,C 0.000} C_DIS
LIN {X 58.511,Y -39.678,Z -109.327,A -90.000,B 90.000,C 0.000} C_DIS
LIN {X 58.383,Y -39.639,Z -109.948,A -90.000,B 90.000,C 0.000} C_DIS
LIN {X 58.330,Y -39.627,Z -110.170,A -90.000,B 90.000,C 0.000} C_DIS
LIN {X 58.123,Y -39.589,Z -110.952,A -90.000,B 90.000,C 0.000} C_DIS
LIN {X 57.688,Y -39.548,Z -112.649,A -90.000,B 90.000,C 0.000} C_DIS
LIN {X 57.634,Y -39.537,Z -112.848,A -90.000,B 90.000,C 0.000} C_DIS
LIN {X 57.528,Y -39.521,Z -113.215,A -90.000,B 90.000,C 0.000} C_DIS
LIN {X 57.284,Y -39.495,Z -113.982,A -90.000,B 90.000,C 0.000} C_DIS
LIN {X 57.170,Y -39.490,Z -114.350,A -90.000,B 90.000,C 0.000} C_DIS
LIN {X 57.140,Y -39.487,Z -114.443,A -90.000,B 90.000,C 0.000} C_DIS
LIN {X 56.949,Y -39.473,Z -114.997,A -90.000,B 90.000,C 0.000} C_DIS
LIN {X 56.559,Y -39.458,Z -116.148,A -90.000,B 90.000,C 0.000} C_DIS
LIN {X 56.392,Y -39.455,Z -116.597,A -90.000,B 90.000,C 0.000} C_DIS
LIN {X 56.094,Y -39.437,Z -117.369,A -90.000,B 90.000,C 0.000} C_DIS
LIN {X 55.945,Y -39.436,Z -117.766,A -90.000,B 90.000,C 0.000} C_DIS
LIN {X 55.887,Y -39.433,Z -117.919,A -90.000,B 90.000,C 0.000} C_DIS
LIN {X 55.715,Y -39.436,Z -118.380,A -90.000,B 90.000,C 0.000} C_DIS
LIN {X 55.641,Y -39.441,Z -118.568,A -90.000,B 90.000,C 0.000} C_DIS
LIN {X 55.524,Y -39.448,Z -118.848,A -90.000,B 90.000,C 0.000} C_DIS
LIN {X 55.467,Y -39.452,Z -118.979,A -90.000,B 90.000,C 0.000} C_DIS
LIN {X 55.119,Y -39.495,Z -119.798,A -90.000,B 90.000,C 0.000} C_DIS
LIN {X 54.978,Y -39.521,Z -120.133,A -90.000,B 90.000,C 0.000} C_DIS
LIN {X 54.714,Y -39.561,Z -120.710,A -90.000,B 90.000,C 0.000} C_DIS
LIN {X 54.147,Y -39.586,Z -121.889,A -90.000,B 90.000,C 0.000} C_DIS
LIN {X 53.945,Y -39.606,Z -122.319,A -90.000,B 90.000,C 0.000} C_DIS
LIN {X 53.806,Y -39.619,Z -122.607,A -90.000,B 90.000,C 0.000} C_DIS
LIN {X 53.756,Y -39.622,Z -122.702,A -90.000,B 90.000,C 0.000} C_DIS
LIN {X 53.549,Y -39.632,Z -123.067,A -90.000,B 90.000,C 0.000} C_DIS
LIN {X 53.215,Y -39.639,Z -123.606,A -90.000,B 90.000,C 0.000} C_DIS
LIN {X 52.067,Y -39.645,Z -125.344,A -90.000,B 90.000,C 0.000} C_DIS
LIN {X 51.311,Y -39.641,Z -126.468,A -90.000,B 90.000,C 0.000} C_DIS
LIN {X 51.166,Y -39.639,Z -126.673,A -90.000,B 90.000,C 0.000} C_DIS
LIN {X 51.019,Y -39.637,Z -126.870,A -90.000,B 90.000,C 0.000} C_DIS
LIN {X 50.830,Y -39.634,Z -127.105,A -90.000,B 90.000,C 0.000} C_DIS
LIN {X 50.682,Y -39.630,Z -127.279,A -90.000,B 90.000,C 0.000} C_DIS
LIN {X 50.630,Y -39.628,Z -127.336,A -90.000,B 90.000,C 0.000} C_DIS
LIN {X 49.512,Y -39.578,Z -128.529,A -90.000,B 90.000,C 0.000} C_DIS
LIN {X 48.227,Y -39.536,Z -129.905,A -90.000,B 90.000,C 0.000} C_DIS
LIN {X 47.995,Y -39.533,Z -130.153,A -90.000,B 90.000,C 0.000} C_DIS
LIN {X 47.794,Y -39.529,Z -130.365,A -90.000,B 90.000,C 0.000} C_DIS
LIN {X 47.658,Y -39.526,Z -130.498,A -90.000,B 90.000,C 0.000} C_DIS
LIN {X 47.376,Y -39.518,Z -130.757,A -90.000,B 90.000,C 0.000} C_DIS
LIN {X 46.588,Y -39.494,Z -131.456,A -90.000,B 90.000,C 0.000} C_DIS
LIN {X 45.293,Y -39.450,Z -132.560,A -90.000,B 90.000,C 0.000} C_DIS
LIN {X 44.471,Y -39.438,Z -133.268,A -90.000,B 90.000,C 0.000} C_DIS
LIN {X 44.171,Y -39.432,Z -133.520,A -90.000,B 90.000,C 0.000} C_DIS
LIN {X 44.080,Y -39.430,Z -133.591,A -90.000,B 90.000,C 0.000} C_DIS
LIN {X 44.044,Y -39.429,Z -133.617,A -90.000,B 90.000,C 0.000} C_DIS
LIN {X 43.629,Y -39.408,Z -133.833,A -90.000,B 90.000,C 0.000} C_DIS
LIN {X 43.333,Y -39.384,Z -133.913,A -90.000,B 90.000,C 0.000} C_DIS
LIN {X 43.189,Y -39.368,Z -133.932,A -90.000,B 90.000,C 0.000} C_DIS
LIN {X 43.075,Y -39.353,Z -133.938,A -90.000,B 90.000,C 0.000} C_DIS
LIN {X 43.039,Y -39.348,Z -133.938,A -90.000,B 90.000,C 0.000} C_DIS
LIN {X 42.801,Y -39.313,Z -133.922,A -90.000,B 90.000,C 0.000} C_DIS
LIN {X 42.768,Y -39.308,Z -133.917,A -90.000,B 90.000,C 0.000} C_DIS
LIN {X 42.768,Y -60.000,Z -133.917,A -90.000,B 90.000,C 0.000} C_DIS
LIN {X 32.783,Y -60.000,Z -153.436,A -90.000,B 90.000,C 0.000} C_DIS
LIN {X 32.783,Y -39.308,Z -153.436,A -90.000,B 90.000,C 0.000} C_DIS
LIN {X 32.820,Y -39.320,Z -153.346,A -90.000,B 90.000,C 0.000} C_DIS
LIN {X 32.973,Y -39.354,Z -152.985,A -90.000,B 90.000,C 0.000} C_DIS
LIN {X 33.068,Y -39.377,Z -152.751,A -90.000,B 90.000,C 0.000} C_DIS
LIN {X 33.258,Y -39.436,Z -152.290,A -90.000,B 90.000,C 0.000} C_DIS
LIN {X 33.454,Y -39.509,Z -151.722,A -90.000,B 90.000,C 0.000} C_DIS
LIN {X 33.592,Y -39.542,Z -151.331,A -90.000,B 90.000,C 0.000} C_DIS
LIN {X 33.741,Y -39.574,Z -150.939,A -90.000,B 90.000,C 0.000} C_DIS
LIN {X 34.021,Y -39.631,Z -150.261,A -90.000,B 90.000,C 0.000} C_DIS
LIN {X 34.232,Y -39.681,Z -149.745,A -90.000,B 90.000,C 0.000} C_DIS
LIN {X 34.373,Y -39.717,Z -149.347,A -90.000,B 90.000,C 0.000} C_DIS
LIN {X 34.451,Y -39.726,Z -149.131,A -90.000,B 90.000,C 0.000} C_DIS
LIN {X 34.558,Y -39.734,Z -148.859,A -90.000,B 90.000,C 0.000} C_DIS
LIN {X 34.637,Y -39.741,Z -148.671,A -90.000,B 90.000,C 0.000} C_DIS
LIN {X 34.784,Y -39.762,Z -148.316,A -90.000,B 90.000,C 0.000} C_DIS
LIN {X 35.098,Y -39.806,Z -147.584,A -90.000,B 90.000,C 0.000} C_DIS
LIN {X 35.367,Y -39.815,Z -146.975,A -90.000,B 90.000,C 0.000} C_DIS
LIN {X 35.480,Y -39.818,Z -146.716,A -90.000,B 90.000,C 0.000} C_DIS
LIN {X 35.552,Y -39.820,Z -146.545,A -90.000,B 90.000,C 0.000} C_DIS
LIN {X 35.729,Y -39.825,Z -146.165,A -90.000,B 90.000,C 0.000} C_DIS
LIN {X 35.945,Y -39.838,Z -145.704,A -90.000,B 90.000,C 0.000} C_DIS
LIN {X 36.054,Y -39.843,Z -145.465,A -90.000,B 90.000,C 0.000} C_DIS
LIN {X 36.405,Y -39.822,Z -144.717,A -90.000,B 90.000,C 0.000} C_DIS
LIN {X 36.590,Y -39.811,Z -144.335,A -90.000,B 90.000,C 0.000} C_DIS
LIN {X 36.633,Y -39.809,Z -144.253,A -90.000,B 90.000,C 0.000} C_DIS
LIN {X 36.951,Y -39.795,Z -143.675,A -90.000,B 90.000,C 0.000} C_DIS
LIN {X 37.050,Y -39.791,Z -143.500,A -90.000,B 90.000,C 0.000} C_DIS
LIN {X 37.482,Y -39.766,Z -142.649,A -90.000,B 90.000,C 0.000} C_DIS
LIN {X 37.663,Y -39.756,Z -142.297,A -90.000,B 90.000,C 0.000} C_DIS
LIN {X 37.794,Y -39.749,Z -142.063,A -90.000,B 90.000,C 0.000} C_DIS
LIN {X 37.901,Y -39.742,Z -141.889,A -90.000,B 90.000,C 0.000} C_DIS
LIN {X 38.073,Y -39.732,Z -141.614,A -90.000,B 90.000,C 0.000} C_DIS
LIN {X 38.433,Y -39.712,Z -141.062,A -90.000,B 90.000,C 0.000} C_DIS
LIN {X 38.865,Y -39.689,Z -140.411,A -90.000,B 90.000,C 0.000} C_DIS
LIN {X 39.071,Y -39.673,Z -140.100,A -90.000,B 90.000,C 0.000} C_DIS
LIN {X 39.384,Y -39.646,Z -139.602,A -90.000,B 90.000,C 0.000} C_DIS
LIN {X 39.562,Y -39.632,Z -139.341,A -90.000,B 90.000,C 0.000} C_DIS
LIN {X 39.616,Y -39.629,Z -139.263,A -90.000,B 90.000,C 0.000} C_DIS
LIN {X 39.898,Y -39.611,Z -138.880,A -90.000,B 90.000,C 0.000} C_DIS
LIN {X 40.253,Y -39.587,Z -138.371,A -90.000,B 90.000,C 0.000} C_DIS
LIN {X 40.942,Y -39.543,Z -137.386,A -90.000,B 90.000,C 0.000} C_DIS
LIN {X 41.064,Y -39.536,Z -137.223,A -90.000,B 90.000,C 0.000} C_DIS
LIN {X 41.105,Y -39.534,Z -137.171,A -90.000,B 90.000,C 0.000} C_DIS
LIN {X 42.209,Y -39.483,Z -135.830,A -90.000,B 90.000,C 0.000} C_DIS
LIN {X 42.099,Y -39.467,Z -135.795,A -90.000,B 90.000,C 0.000} C_DIS
LIN {X 42.016,Y -39.454,Z -135.765,A -90.000,B 90.000,C 0.000} C_DIS
LIN {X 41.902,Y -39.436,Z -135.716,A -90.000,B 90.000,C 0.000} C_DIS
LIN {X 41.752,Y -39.407,Z -135.637,A -90.000,B 90.000,C 0.000} C_DIS
LIN {X 41.731,Y -39.403,Z -135.625,A -90.000,B 90.000,C 0.000} C_DIS
LIN {X 41.533,Y -39.359,Z -135.490,A -90.000,B 90.000,C 0.000} C_DIS
LIN {X 41.442,Y -39.337,Z -135.414,A -90.000,B 90.000,C 0.000} C_DIS
LIN {X 41.334,Y -39.308,Z -135.311,A -90.000,B 90.000,C 0.000} C_DIS
LIN {X 41.334,Y -60.000,Z -135.311,A -90.000,B 90.000,C 0.000} C_DIS
LIN {X 30.790,Y -60.000,Z -153.607,A -90.000,B 90.000,C 0.000} C_DIS
LIN {X 30.790,Y -39.308,Z -153.607,A -90.000,B 90.000,C 0.000} C_DIS
LIN {X 30.784,Y -39.347,Z -153.367,A -90.000,B 90.000,C 0.000} C_DIS
LIN {X 30.792,Y -39.363,Z -153.251,A -90.000,B 90.000,C 0.000} C_DIS
LIN {X 30.798,Y -39.371,Z -153.193,A -90.000,B 90.000,C 0.000} C_DIS
LIN {X 30.935,Y -39.432,Z -152.681,A -90.000,B 90.000,C 0.000} C_DIS
LIN {X 31.130,Y -39.487,Z -152.219,A -90.000,B 90.000,C 0.000} C_DIS
LIN {X 31.228,Y -39.514,Z -151.978,A -90.000,B 90.000,C 0.000} C_DIS
LIN {X 31.385,Y -39.549,Z -151.596,A -90.000,B 90.000,C 0.000} C_DIS
LIN {X 31.592,Y -39.605,Z -150.997,A -90.000,B 90.000,C 0.000} C_DIS
LIN {X 31.718,Y -39.633,Z -150.640,A -90.000,B 90.000,C 0.000} C_DIS
LIN {X 31.805,Y -39.651,Z -150.409,A -90.000,B 90.000,C 0.000} C_DIS
LIN {X 31.888,Y -39.664,Z -150.191,A -90.000,B 90.000,C 0.000} C_DIS
LIN {X 32.273,Y -39.720,Z -149.255,A -90.000,B 90.000,C 0.000} C_DIS
LIN {X 32.361,Y -39.730,Z -149.037,A -90.000,B 90.000,C 0.000} C_DIS
LIN {X 32.569,Y -39.748,Z -148.454,A -90.000,B 90.000,C 0.000} C_DIS
LIN {X 32.728,Y -39.760,Z -148.052,A -90.000,B 90.000,C 0.000} C_DIS
LIN {X 32.804,Y -39.764,Z -147.871,A -90.000,B 90.000,C 0.000} C_DIS
LIN {X 33.027,Y -39.764,Z -147.338,A -90.000,B 90.000,C 0.000} C_DIS
LIN {X 33.270,Y -39.763,Z -146.775,A -90.000,B 90.000,C 0.000} C_DIS
LIN {X 33.642,Y -39.763,Z -145.929,A -90.000,B 90.000,C 0.000} C_DIS
LIN {X 33.739,Y -39.758,Z -145.702,A -90.000,B 90.000,C 0.000} C_DIS
LIN {X 34.203,Y -39.730,Z -144.712,A -90.000,B 90.000,C 0.000} C_DIS
LIN {X 34.563,Y -39.697,Z -143.943,A -90.000,B 90.000,C 0.000} C_DIS
LIN {X 34.815,Y -39.668,Z -143.426,A -90.000,B 90.000,C 0.000} C_DIS
LIN {X 34.884,Y -39.661,Z -143.293,A -90.000,B 90.000,C 0.000} C_DIS
LIN {X 35.214,Y -39.629,Z -142.696,A -90.000,B 90.000,C 0.000} C_DIS
LIN {X 35.292,Y -39.622,Z -142.560,A -90.000,B 90.000,C 0.000} C_DIS
LIN {X 35.488,Y -39.601,Z -142.176,A -90.000,B 90.000,C 0.000} C_DIS
LIN {X 35.893,Y -39.535,Z -141.393,A -90.000,B 90.000,C 0.000} C_DIS
LIN {X 36.093,Y -39.507,Z -141.039,A -90.000,B 90.000,C 0.000} C_DIS
LIN {X 36.366,Y -39.474,Z -140.604,A -90.000,B 90.000,C 0.000} C_DIS
LIN {X 36.779,Y -39.428,Z -139.975,A -90.000,B 90.000,C 0.000} C_DIS
LIN {X 37.400,Y -39.363,Z -139.045,A -90.000,B 90.000,C 0.000} C_DIS
LIN {X 37.744,Y -39.322,Z -138.505,A -90.000,B 90.000,C 0.000} C_DIS
LIN {X 37.868,Y -39.308,Z -138.324,A -90.000,B 90.000,C 0.000} C_DIS
LIN {X 37.868,Y -60.000,Z -138.324,A -90.000,B 90.000,C 0.000} C_DIS
LIN {X 28.803,Y -60.000,Z -153.833,A -90.000,B 90.000,C 0.000} C_DIS
LIN {X 28.803,Y -39.308,Z -153.833,A -90.000,B 90.000,C 0.000} C_DIS
LIN {X 28.798,Y -39.315,Z -153.784,A -90.000,B 90.000,C 0.000} C_DIS
LIN {X 28.791,Y -39.330,Z -153.659,A -90.000,B 90.000,C 0.000} C_DIS
LIN {X 28.785,Y -39.361,Z -153.417,A -90.000,B 90.000,C 0.000} C_DIS
LIN {X 28.786,Y -39.376,Z -153.290,A -90.000,B 90.000,C 0.000} C_DIS
LIN {X 28.797,Y -39.393,Z -153.117,A -90.000,B 90.000,C 0.000} C_DIS
LIN {X 28.807,Y -39.402,Z -153.007,A -90.000,B 90.000,C 0.000} C_DIS
LIN {X 28.828,Y -39.415,Z -152.854,A -90.000,B 90.000,C 0.000} C_DIS
LIN {X 28.856,Y -39.426,Z -152.720,A -90.000,B 90.000,C 0.000} C_DIS
LIN {X 28.903,Y -39.441,Z -152.541,A -90.000,B 90.000,C 0.000} C_DIS
LIN {X 29.001,Y -39.466,Z -152.170,A -90.000,B 90.000,C 0.000} C_DIS
LIN {X 29.053,Y -39.477,Z -152.006,A -90.000,B 90.000,C 0.000} C_DIS
LIN {X 29.091,Y -39.484,Z -151.907,A -90.000,B 90.000,C 0.000} C_DIS
LIN {X 29.277,Y -39.518,Z -151.467,A -90.000,B 90.000,C 0.000} C_DIS
LIN {X 29.513,Y -39.561,Z -150.890,A -90.000,B 90.000,C 0.000} C_DIS
LIN {X 29.718,Y -39.602,Z -150.297,A -90.000,B 90.000,C 0.000} C_DIS
LIN {X 29.863,Y -39.630,Z -149.891,A -90.000,B 90.000,C 0.000} C_DIS
LIN {X 30.038,Y -39.643,Z -149.430,A -90.000,B 90.000,C 0.000} C_DIS
LIN {X 30.232,Y -39.645,Z -148.961,A -90.000,B 90.000,C 0.000} C_DIS
LIN {X 30.494,Y -39.645,Z -148.323,A -90.000,B 90.000,C 0.000} C_DIS
LIN {X 30.689,Y -39.632,Z -147.781,A -90.000,B 90.000,C 0.000} C_DIS
LIN {X 30.874,Y -39.623,Z -147.315,A -90.000,B 90.000,C 0.000} C_DIS
LIN {X 31.195,Y -39.610,Z -146.551,A -90.000,B 90.000,C 0.000} C_DIS
LIN {X 31.412,Y -39.601,Z -146.049,A -90.000,B 90.000,C 0.000} C_DIS
LIN {X 31.560,Y -39.587,Z -145.713,A -90.000,B 90.000,C 0.000} C_DIS
LIN {X 31.817,Y -39.543,Z -145.139,A -90.000,B 90.000,C 0.000} C_DIS
LIN {X 31.938,Y -39.523,Z -144.865,A -90.000,B 90.000,C 0.000} C_DIS
LIN {X 32.055,Y -39.505,Z -144.618,A -90.000,B 90.000,C 0.000} C_DIS
LIN {X 32.782,Y -39.367,Z -143.096,A -90.000,B 90.000,C 0.000} C_DIS
LIN {X 33.035,Y -39.322,Z -142.580,A -90.000,B 90.000,C 0.000} C_DIS
LIN {X 33.116,Y -39.308,Z -142.427,A -90.000,B 90.000,C 0.000} C_DIS
LIN {X 33.116,Y -60.000,Z -142.427,A -90.000,B 90.000,C 0.000} C_DIS
LIN {X 26.862,Y -60.000,Z -152.503,A -90.000,B 90.000,C 0.000} C_DIS
LIN {X 26.862,Y -39.308,Z -152.503,A -90.000,B 90.000,C 0.000} C_DIS
LIN {X 26.882,Y -39.317,Z -152.402,A -90.000,B 90.000,C 0.000} C_DIS
LIN {X 26.926,Y -39.327,Z -152.204,A -90.000,B 90.000,C 0.000} C_DIS
LIN {X 27.014,Y -39.339,Z -151.875,A -90.000,B 90.000,C 0.000} C_DIS
LIN {X 27.074,Y -39.340,Z -151.650,A -90.000,B 90.000,C 0.000} C_DIS
LIN {X 27.117,Y -39.342,Z -151.508,A -90.000,B 90.000,C 0.000} C_DIS
LIN {X 27.150,Y -39.343,Z -151.403,A -90.000,B 90.000,C 0.000} C_DIS
LIN {X 27.207,Y -39.346,Z -151.246,A -90.000,B 90.000,C 0.000} C_DIS
LIN {X 27.256,Y -39.349,Z -151.123,A -90.000,B 90.000,C 0.000} C_DIS
LIN {X 27.444,Y -39.362,Z -150.681,A -90.000,B 90.000,C 0.000} C_DIS
LIN {X 27.653,Y -39.375,Z -150.176,A -90.000,B 90.000,C 0.000} C_DIS
LIN {X 27.851,Y -39.384,Z -149.614,A -90.000,B 90.000,C 0.000} C_DIS
LIN {X 28.033,Y -39.393,Z -149.117,A -90.000,B 90.000,C 0.000} C_DIS
LIN {X 28.078,Y -39.395,Z -148.999,A -90.000,B 90.000,C 0.000} C_DIS
LIN {X 28.204,Y -39.395,Z -148.673,A -90.000,B 90.000,C 0.000} C_DIS
LIN {X 28.346,Y -39.394,Z -148.329,A -90.000,B 90.000,C 0.000} C_DIS
LIN {X 28.430,Y -39.388,Z -148.128,A -90.000,B 90.000,C 0.000} C_DIS
LIN {X 28.543,Y -39.375,Z -147.856,A -90.000,B 90.000,C 0.000} C_DIS
LIN {X 28.646,Y -39.357,Z -147.614,A -90.000,B 90.000,C 0.000} C_DIS
LIN {X 28.853,Y -39.308,Z -147.058,A -90.000,B 90.000,C 0.000} C_DIS
LIN {X 28.853,Y -60.000,Z -147.058,A -90.000,B 90.000,C 0.000} C_DIS
LIN {X 61.050,Y -60.000,Z -106.438,A -90.000,B 90.000,C 0.000} C_DIS
LIN {X 61.050,Y -39.411,Z -106.438,A -90.000,B 90.000,C 0.000} C_DIS
LIN {X 61.208,Y -39.431,Z -106.097,A -90.000,B 90.000,C 0.000} C_DIS
LIN {X 61.223,Y -39.433,Z -106.059,A -90.000,B 90.000,C 0.000} C_DIS
LIN {X 61.301,Y -39.443,Z -105.872,A -90.000,B 90.000,C 0.000} C_DIS
LIN {X 61.409,Y -39.458,Z -105.609,A -90.000,B 90.000,C 0.000} C_DIS
LIN {X 61.623,Y -39.487,Z -105.079,A -90.000,B 90.000,C 0.000} C_DIS
LIN {X 61.768,Y -39.520,Z -104.645,A -90.000,B 90.000,C 0.000} C_DIS
LIN {X 62.117,Y -39.614,Z -103.600,A -90.000,B 90.000,C 0.000} C_DIS
LIN {X 62.277,Y -39.670,Z -102.902,A -90.000,B 90.000,C 0.000} C_DIS
LIN {X 62.413,Y -39.714,Z -102.368,A -90.000,B 90.000,C 0.000} C_DIS
LIN {X 62.437,Y -39.732,Z -102.173,A -90.000,B 90.000,C 0.000} C_DIS
LIN {X 62.221,Y -39.760,Z -101.541,A -90.000,B 90.000,C 0.000} C_DIS
LIN {X 62.082,Y -39.767,Z -101.281,A -90.000,B 90.000,C 0.000} C_DIS
LIN {X 61.701,Y -39.859,Z -100.592,A -90.000,B 90.000,C 0.000} C_DIS
LIN {X 61.547,Y -39.881,Z -100.306,A -90.000,B 90.000,C 0.000} C_DIS
LIN {X 61.556,Y -39.843,Z -100.739,A -90.000,B 90.000,C 0.000} C_DIS
LIN {X 61.565,Y -39.771,Z -101.316,A -90.000,B 90.000,C 0.000} C_DIS
LIN {X 61.559,Y -39.735,Z -101.602,A -90.000,B 90.000,C 0.000} C_DIS
LIN {X 61.539,Y -39.712,Z -101.970,A -90.000,B 90.000,C 0.000} C_DIS
LIN {X 61.512,Y -39.695,Z -102.257,A -90.000,B 90.000,C 0.000} C_DIS
LIN {X 61.416,Y -39.645,Z -103.061,A -90.000,B 90.000,C 0.000} C_DIS
LIN {X 61.342,Y -39.586,Z -103.637,A -90.000,B 90.000,C 0.000} C_DIS
LIN {X 61.234,Y -39.498,Z -104.493,A -90.000,B 90.000,C 0.000} C_DIS
LIN {X 61.213,Y -39.486,Z -104.676,A -90.000,B 90.000,C 0.000} C_DIS
LIN {X 61.205,Y -39.479,Z -104.788,A -90.000,B 90.000,C 0.000} C_DIS
LIN {X 61.143,Y -39.441,Z -105.755,A -90.000,B 90.000,C 0.000} C_DIS
LIN {X 61.132,Y -39.436,Z -105.865,A -90.000,B 90.000,C 0.000} C_DIS
LIN {X 61.091,Y -39.422,Z -106.197,A -90.000,B 90.000,C 0.000} C_DIS
LIN {X 61.066,Y -39.415,Z -106.352,A -90.000,B 90.000,C 0.000} C_DIS
LIN {X 61.050,Y -39.411,Z -106.438,A -90.000,B 90.000,C 0.000} C_DIS
LIN {X 61.050,Y -60.000,Z -106.438,A -90.000,B 90.000,C 0.000} C_DIS
LIN {X 58.752,Y -60.000,Z -88.665,A -90.000,B 90.000,C 0.000} C_DIS
LIN {X 58.752,Y -40.195,Z -88.665,A -90.000,B 90.000,C 0.000} C_DIS
LIN {X 58.751,Y -40.155,Z -88.144,A -90.000,B 90.000,C 0.000} C_DIS
LIN {X 58.754,Y -40.139,Z -87.949,A -90.000,B 90.000,C 0.000} C_DIS
LIN {X 58.769,Y -40.131,Z -87.595,A -90.000,B 90.000,C 0.000} C_DIS
LIN {X 58.795,Y -40.120,Z -87.130,A -90.000,B 90.000,C 0.000} C_DIS
LIN {X 58.802,Y -40.116,Z -87.012,A -90.000,B 90.000,C 0.000} C_DIS
LIN {X 58.803,Y -40.116,Z -87.000,A -90.000,B 90.000,C 0.000} C_DIS
LIN {X 58.810,Y -40.108,Z -86.868,A -90.000,B 90.000,C 0.000} C_DIS
LIN {X 58.842,Y -40.058,Z -86.001,A -90.000,B 90.000,C 0.000} C_DIS
LIN {X 58.832,Y -40.014,Z -85.181,A -90.000,B 90.000,C 0.000} C_DIS
LIN {X 58.827,Y -40.002,Z -84.778,A -90.000,B 90.000,C 0.000} C_DIS
LIN {X 58.824,Y -40.003,Z -84.525,A -90.000,B 90.000,C 0.000} C_DIS
LIN {X 58.830,Y -40.003,Z -84.300,A -90.000,B 90.000,C 0.000} C_DIS
LIN {X 58.845,Y -40.016,Z -83.871,A -90.000,B 90.000,C 0.000} C_DIS
LIN {X 58.853,Y -40.019,Z -83.751,A -90.000,B 90.000,C 0.000} C_DIS
LIN {X 58.847,Y -40.033,Z -83.332,A -90.000,B 90.000,C 0.000} C_DIS
LIN {X 58.829,Y -40.054,Z -82.724,A -90.000,B 90.000,C 0.000} C_DIS
LIN {X 58.818,Y -40.059,Z -82.602,A -90.000,B 90.000,C 0.000} C_DIS
LIN {X 58.773,Y -40.066,Z -82.065,A -90.000,B 90.000,C 0.000} C_DIS
LIN {X 58.743,Y -40.109,Z -81.733,A -90.000,B 90.000,C 0.000} C_DIS
LIN {X 58.679,Y -40.137,Z -81.515,A -90.000,B 90.000,C 0.000} C_DIS
LIN {X 57.987,Y -40.119,Z -81.664,A -90.000,B 90.000,C 0.000} C_DIS
LIN {X 57.673,Y -40.138,Z -81.735,A -90.000,B 90.000,C 0.000} C_DIS
LIN {X 57.394,Y -40.155,Z -81.792,A -90.000,B 90.000,C 0.000} C_DIS
LIN {X 56.911,Y -40.207,Z -81.894,A -90.000,B 90.000,C 0.000} C_DIS
LIN {X 56.284,Y -40.272,Z -82.125,A -90.000,B 90.000,C 0.000} C_DIS
LIN {X 55.514,Y -40.351,Z -82.392,A -90.000,B 90.000,C 0.000} C_DIS
LIN {X 55.132,Y -40.391,Z -82.528,A -90.000,B 90.000,C 0.000} C_DIS
LIN {X 54.995,Y -40.405,Z -82.577,A -90.000,B 90.000,C 0.000} C_DIS
